C05458=1043.474,385.726,371.742,173.657,43.122,158.451
C05459=1043.465,385.481,371.783,173.649,43.117,158.449
C05460=1043.457,385.234,371.825,173.642,43.112,158.447
C05461=1043.448,384.988,371.867,173.634,43.107,158.445
C05462=1043.439,384.741,371.909,173.627,43.102,158.444
C05463=1043.432,384.495,371.951,173.621,43.097,158.442
C05464=1043.423,384.249,371.992,173.614,43.091,158.440
C05465=1043.414,384.003,372.034,173.606,43.086,158.438
C05466=1043.406,383.757,372.076,173.599,43.082,158.436
C05467=1043.397,383.510,372.118,173.592,43.077,158.435
C05468=1043.389,383.263,372.159,173.584,43.071,158.433
C05469=1043.380,383.018,372.200,173.577,43.066,158.431
C05470=1043.371,382.771,372.242,173.571,43.061,158.429
C05471=1043.363,382.524,372.284,173.564,43.056,158.427
C05472=1043.355,382.278,372.325,173.557,43.052,158.426
C05473=1043.346,382.032,372.367,173.549,43.047,158.424
C05474=1043.338,381.786,372.407,173.542,43.042,158.422
C05475=1043.330,381.539,372.450,173.536,43.037,158.420
C05476=1043.322,381.293,372.491,173.529,43.032,158.419
C05477=1043.313,381.046,372.532,173.521,43.027,158.417
C05478=1043.305,380.801,372.573,173.514,43.022,158.415
C05479=1043.297,380.553,372.615,173.507,43.017,158.413
C05480=1043.289,380.308,372.656,173.501,43.012,158.412
C05481=1043.280,380.061,372.697,173.494,43.007,158.410
C05482=1043.272,379.814,372.738,173.486,43.002,158.408
C05483=1043.264,379.569,372.779,173.480,42.997,158.406
C05484=1043.256,379.321,372.821,173.473,42.992,158.405
C05485=1043.248,379.075,372.861,173.466,42.988,158.403
C05486=1043.239,378.829,372.903,173.460,42.983,158.401
C05487=1043.231,378.582,372.944,173.453,42.978,158.400
C05488=1043.223,378.336,372.984,173.446,42.974,158.398
C05489=1043.214,378.089,373.025,173.438,42.969,158.396
C05490=1043.205,377.843,373.065,173.432,42.964,158.395
C05491=1043.197,377.596,373.106,173.425,42.959,158.393
C05492=1043.189,377.350,373.147,173.418,42.955,158.391
C05493=1043.176,376.988,373.207,173.409,42.948,158.389
C05494=1043.165,376.627,373.267,173.399,42.941,158.386
C05495=1043.153,376.264,373.326,173.389,42.934,158.384
C05496=1043.140,375.903,373.386,173.379,42.928,158.382
C05497=1043.132,375.656,373.426,173.373,42.923,158.380
C05498=1043.124,375.410,373.467,173.366,42.919,158.378
C05499=1043.116,375.163,373.507,173.360,42.914,158.377
C05500=1043.107,374.916,373.548,173.353,42.909,158.375
C05501=1043.099,374.670,373.589,173.346,42.905,158.373
C05502=1043.092,374.423,373.629,173.340,42.900,158.372
C05503=1043.083,374.177,373.669,173.333,42.896,158.370
C05504=1043.075,373.931,373.710,173.327,42.891,158.369
C05505=1043.067,373.684,373.749,173.320,42.887,158.367
C05506=1043.058,373.437,373.790,173.314,42.882,158.365
C05507=1043.051,373.190,373.830,173.307,42.877,158.364
C05508=1043.043,372.944,373.871,173.301,42.873,158.362
C05509=1043.035,372.697,373.912,173.294,42.869,158.361
C05510=1043.026,372.451,373.951,173.288,42.864,158.359
C05511=1043.018,372.205,373.992,173.281,42.860,158.358
C05512=1043.010,371.958,374.032,173.275,42.855,158.356
C05513=1043.003,371.711,374.071,173.268,42.851,158.354
C05514=1042.995,371.465,374.112,173.262,42.846,158.353
C05515=1042.987,371.218,374.152,173.257,42.842,158.351
C05516=1042.978,370.972,374.192,173.250,42.838,158.350
C05517=1042.971,370.725,374.232,173.244,42.833,158.348
C05518=1042.963,370.478,374.272,173.237,42.829,158.347
C05519=1042.954,370.231,374.311,173.231,42.824,158.345
C05520=1042.947,369.984,374.351,173.224,42.821,158.344
C05521=1042.939,369.738,374.392,173.218,42.816,158.342
C05522=1042.930,369.491,374.431,173.212,42.812,158.341
C05523=1042.922,369.245,374.471,173.205,42.808,158.339
C05524=1042.914,368.998,374.510,173.199,42.803,158.338
C05525=1042.906,368.751,374.550,173.193,42.799,158.336
C05526=1042.898,368.504,374.590,173.187,42.795,158.335
C05527=1042.890,368.258,374.629,173.181,42.791,158.333
C05528=1042.882,368.011,374.669,173.174,42.786,158.332
C05529=1042.874,367.764,374.709,173.168,42.782,158.330
C05530=1042.866,367.518,374.748,173.162,42.778,158.329
C05531=1042.858,367.271,374.788,173.156,42.774,158.327
C05532=1042.850,367.024,374.826,173.150,42.769,158.326
C05533=1042.842,366.777,374.866,173.143,42.766,158.325
C05534=1042.834,366.531,374.905,173.137,42.762,158.323
C05535=1042.826,366.284,374.945,173.131,42.757,158.322
C05536=1042.818,366.038,374.984,173.126,42.753,158.320
C05537=1042.811,365.790,375.024,173.119,42.749,158.319
C05538=1042.803,365.544,375.063,173.113,42.745,158.317
C05539=1042.795,365.297,375.103,173.107,42.741,158.316
C05540=1042.787,365.051,375.142,173.101,42.737,158.314
C05541=1042.780,364.803,375.181,173.095,42.732,158.313
C05542=1042.771,364.557,375.220,173.089,42.728,158.312
C05543=1042.764,364.310,375.259,173.083,42.724,158.310
C05544=1042.756,364.063,375.298,173.077,42.721,158.309
C05545=1042.748,363.816,375.338,173.071,42.717,158.307
C05546=1042.741,363.570,375.377,173.065,42.713,158.306
C05547=1042.733,363.323,375.416,173.059,42.708,158.304
C05548=1042.725,363.076,375.455,173.054,42.704,158.303
C05549=1042.714,362.733,375.509,173.045,42.698,158.301
C05550=1042.704,362.392,375.564,173.037,42.693,158.299
C05551=1042.693,362.050,375.617,173.029,42.688,158.297
C05552=1042.682,361.707,375.671,173.020,42.682,158.295
C05553=1042.674,361.461,375.709,173.014,42.678,158.294
C05554=1042.666,361.214,375.749,173.009,42.674,158.293
C05555=1042.658,360.967,375.787,173.003,42.670,158.291
C05556=1042.651,360.720,375.826,172.998,42.667,158.290
C05557=1042.643,360.473,375.865,172.992,42.663,158.289
C05558=1042.635,360.226,375.903,172.985,42.659,158.287
C05559=1042.627,359.979,375.942,172.979,42.655,158.286
C05560=1042.619,359.733,375.981,172.974,42.651,158.285
C05561=1042.612,359.486,376.020,172.968,42.647,158.283
C05562=1042.604,359.239,376.058,172.963,42.643,158.282
C05563=1042.596,358.992,376.097,172.957,42.639,158.281
C05564=1042.588,358.745,376.135,172.951,42.636,158.279
C05565=1042.580,358.498,376.174,172.946,42.632,158.278
C05566=1042.573,358.252,376.212,172.939,42.628,158.277
C05567=1042.565,358.004,376.250,172.934,42.625,158.275
C05568=1042.558,357.757,376.289,172.928,42.621,158.274
C05569=1042.550,357.510,376.327,172.922,42.617,158.273
C05570=1042.542,357.263,376.365,172.917,42.613,158.271
C05571=1042.535,357.017,376.404,172.911,42.610,158.270
C05572=1042.527,356.770,376.442,172.906,42.606,158.269
C05573=1042.519,356.523,376.480,172.900,42.602,158.268
C05574=1042.511,356.275,376.518,172.894,42.598,158.266
C05575=1042.504,356.029,376.557,172.889,42.595,158.265
C05576=1042.496,355.782,376.595,172.883,42.591,158.264
C05577=1042.488,355.534,376.633,172.878,42.587,158.262
C05578=1042.481,355.288,376.671,172.872,42.584,158.261
C05579=1042.473,355.041,376.709,172.867,42.580,158.260
C05580=1042.465,354.793,376.747,172.861,42.576,158.259
C05581=1042.458,354.547,376.785,172.856,42.573,158.257
C05582=1042.451,354.300,376.823,172.850,42.569,158.256
C05583=1042.442,354.053,376.861,172.844,42.565,158.255
C05584=1042.435,353.805,376.899,172.839,42.562,158.254
C05585=1042.428,353.559,376.937,172.834,42.558,158.252
C05586=1042.420,353.312,376.974,172.828,42.555,158.251
C05587=1042.412,353.065,377.013,172.822,42.551,158.250
C05588=1042.404,352.818,377.050,172.817,42.547,158.249
C05589=1042.397,352.571,377.088,172.811,42.544,158.247
C05590=1042.390,352.324,377.126,172.806,42.540,158.246
C05591=1042.382,352.077,377.164,172.801,42.537,158.245
C05592=1042.374,351.829,377.202,172.795,42.533,158.244
C05593=1042.367,351.583,377.240,172.789,42.529,158.242
C05594=1042.360,351.335,377.277,172.784,42.526,158.241
C05595=1042.352,351.088,377.315,172.778,42.522,158.240
C05596=1042.345,350.842,377.353,172.773,42.519,158.239
C05597=1042.337,350.595,377.390,172.769,42.515,158.238
C05598=1042.330,350.348,377.428,172.763,42.512,158.236
C05599=1042.322,350.100,377.465,172.758,42.508,158.235
C05600=1042.315,349.853,377.503,172.752,42.505,158.234
C05601=1042.307,349.606,377.540,172.747,42.501,158.233
C05602=1042.299,349.359,377.577,172.741,42.498,158.232
C05603=1042.292,349.112,377.615,172.736,42.495,158.231
C05604=1042.285,348.865,377.652,172.730,42.492,158.229
C05605=1042.274,348.529,377.703,172.723,42.486,158.228
C05606=1042.264,348.192,377.754,172.717,42.482,158.226
C05607=1042.254,347.857,377.805,172.710,42.477,158.225
C05608=1042.243,347.519,377.856,172.702,42.473,158.223
C05609=1042.236,347.272,377.893,172.697,42.469,158.222
C05610=1042.228,347.025,377.930,172.692,42.466,158.221
C05611=1042.221,346.778,377.968,172.687,42.463,158.220
C05612=1042.214,346.530,378.005,172.681,42.460,158.218
C05613=1042.206,346.284,378.041,172.676,42.456,158.217
C05614=1042.199,346.037,378.079,172.671,42.452,158.216
C05615=1042.191,345.790,378.116,172.666,42.450,158.215
C05616=1042.184,345.543,378.153,172.661,42.446,158.214
C05617=1042.177,345.295,378.190,172.655,42.443,158.213
C05618=1042.169,345.049,378.227,172.650,42.440,158.212
C05619=1042.162,344.802,378.264,172.645,42.436,158.210
C05620=1042.154,344.554,378.301,172.640,42.433,158.209
C05621=1042.147,344.307,378.338,172.635,42.430,158.208
C05622=1042.139,344.059,378.374,172.629,42.427,158.207
C05623=1042.132,343.812,378.412,172.625,42.423,158.206
C05624=1042.125,343.565,378.449,172.620,42.420,158.205
C05625=1042.118,343.318,378.485,172.614,42.417,158.204
C05626=1042.110,343.071,378.523,172.609,42.414,158.203
C05627=1042.103,342.824,378.559,172.605,42.410,158.201
C05628=1042.096,342.576,378.596,172.599,42.407,158.200
C05629=1042.088,342.329,378.633,172.594,42.404,158.199
C05630=1042.082,342.082,378.669,172.590,42.401,158.198
C05631=1042.074,341.835,378.706,172.585,42.398,158.197
C05632=1042.067,341.588,378.743,172.579,42.394,158.196
C05633=1042.059,341.340,378.779,172.574,42.391,158.195
C05634=1042.051,341.093,378.816,172.570,42.388,158.194
C05635=1042.044,340.846,378.853,172.564,42.385,158.193
C05636=1042.037,340.599,378.889,172.559,42.382,158.192
C05637=1042.029,340.351,378.925,172.555,42.379,158.191
C05638=1042.021,340.105,378.962,172.549,42.376,158.190
C05639=1042.014,339.857,378.999,172.544,42.372,158.188
C05640=1042.007,339.610,379.035,172.540,42.369,158.187
C05641=1042.000,339.363,379.071,172.535,42.366,158.186
C05642=1041.993,339.115,379.108,172.529,42.363,158.185
C05643=1041.986,338.868,379.143,172.525,42.360,158.184
C05644=1041.978,338.621,379.180,172.520,42.357,158.183
C05645=1041.970,338.374,379.217,172.514,42.354,158.182
C05646=1041.964,338.127,379.253,172.510,42.351,158.181
C05647=1041.956,337.879,379.289,172.505,42.348,158.180
C05648=1041.948,337.632,379.325,172.500,42.345,158.179
C05649=1041.942,337.385,379.362,172.495,42.342,158.178
C05650=1041.934,337.137,379.398,172.490,42.339,158.177
C05651=1041.927,336.890,379.434,172.486,42.336,158.176
C05652=1041.919,336.643,379.470,172.481,42.333,158.175
C05653=1041.913,336.396,379.507,172.476,42.330,158.174
C05654=1041.906,336.148,379.542,172.471,42.327,158.173
C05655=1041.898,335.901,379.578,172.466,42.324,158.172
C05656=1041.890,335.653,379.615,172.462,42.321,158.171
C05657=1041.884,335.406,379.651,172.457,42.318,158.170
C05658=1041.876,335.159,379.687,172.452,42.315,158.169
C05659=1041.869,334.912,379.723,172.447,42.312,158.168
C05660=1041.862,334.664,379.759,172.442,42.309,158.167
C05661=1041.852,334.324,379.808,172.435,42.305,158.165
C05662=1041.842,333.984,379.857,172.430,42.301,158.164
C05663=1041.832,333.644,379.906,172.423,42.297,158.163
C05664=1041.822,333.304,379.956,172.416,42.293,158.161
C05665=1041.815,333.057,379.991,172.411,42.290,158.160
C05666=1041.808,332.809,380.027,172.407,42.287,158.159
C05667=1041.800,332.563,380.063,172.402,42.284,158.158
C05668=1041.793,332.315,380.098,172.398,42.281,158.157
C05669=1041.786,332.068,380.134,172.393,42.278,158.156
C05670=1041.778,331.820,380.170,172.388,42.275,158.155
C05671=1041.772,331.573,380.205,172.383,42.273,158.154
C05672=1041.764,331.325,380.241,172.379,42.270,158.153
C05673=1041.757,331.078,380.277,172.374,42.267,158.152
C05674=1041.750,330.831,380.312,172.370,42.264,158.152
C05675=1041.743,330.583,380.348,172.365,42.261,158.151
C05676=1041.736,330.336,380.383,172.360,42.258,158.150
C05677=1041.728,330.089,380.420,172.355,42.256,158.149
C05678=1041.722,329.841,380.455,172.351,42.253,158.148
C05679=1041.715,329.594,380.490,172.346,42.250,158.147
C05680=1041.707,329.346,380.526,172.342,42.247,158.146
C05681=1041.700,329.099,380.561,172.338,42.244,158.145
C05682=1041.693,328.852,380.596,172.333,42.241,158.144
C05683=1041.685,328.604,380.631,172.328,42.239,158.143
C05684=1041.678,328.357,380.667,172.323,42.236,158.142
C05685=1041.670,328.109,380.702,172.319,42.233,158.141
C05686=1041.663,327.862,380.737,172.314,42.231,158.140
C05687=1041.656,327.615,380.772,172.310,42.228,158.139
C05688=1041.649,327.367,380.807,172.305,42.225,158.138
C05689=1041.642,327.120,380.842,172.301,42.223,158.137
C05690=1041.634,326.873,380.877,172.296,42.220,158.136
C05691=1041.627,326.624,380.912,172.292,42.217,158.136
C05692=1041.619,326.377,380.947,172.287,42.215,158.135
C05693=1041.613,326.130,380.982,172.283,42.212,158.134
C05694=1041.605,325.882,381.017,172.279,42.209,158.133
C05695=1041.598,325.635,381.052,172.274,42.207,158.132
C05696=1041.591,325.388,381.087,172.269,42.204,158.131
C05697=1041.584,325.140,381.122,172.264,42.201,158.130
C05698=1041.576,324.892,381.157,172.260,42.199,158.129
C05699=1041.569,324.645,381.192,172.256,42.196,158.128
C05700=1041.562,324.398,381.227,172.251,42.193,158.127
C05701=1041.554,324.151,381.261,172.247,42.191,158.127
C05702=1041.548,323.903,381.296,172.242,42.188,158.126
C05703=1041.541,323.655,381.331,172.238,42.185,158.125
C05704=1041.533,323.408,381.366,172.234,42.183,158.124
C05705=1041.526,323.160,381.401,172.229,42.180,158.123
C05706=1041.519,322.913,381.436,172.225,42.178,158.122
C05707=1041.512,322.665,381.470,172.221,42.175,158.121
C05708=1041.505,322.418,381.504,172.216,42.172,158.120
C05709=1041.497,322.170,381.540,172.212,42.170,158.119
C05710=1041.490,321.923,381.575,172.208,42.167,158.119
C05711=1041.483,321.675,381.609,172.203,42.165,158.118
C05712=1041.476,321.428,381.643,172.199,42.162,158.117
C05713=1041.469,321.181,381.679,172.195,42.160,158.116
C05714=1041.462,320.933,381.712,172.189,42.157,158.115
C05715=1041.455,320.686,381.748,172.185,42.154,158.114
C05716=1041.448,320.438,381.781,172.181,42.152,158.113
C05717=1041.438,320.094,381.831,172.175,42.148,158.112
C05718=1041.428,319.749,381.879,172.170,42.145,158.111
C05719=1041.418,319.404,381.927,172.163,42.141,158.110
C05720=1041.409,319.059,381.975,172.157,42.138,158.108
C05721=1041.402,318.811,382.009,172.153,42.135,158.108
C05722=1041.395,318.564,382.044,172.149,42.133,158.107
C05723=1041.388,318.316,382.078,172.145,42.130,158.106
C05724=1041.381,318.069,382.113,172.140,42.128,158.105
C05725=1041.375,317.822,382.146,172.136,42.125,158.104
C05726=1041.368,317.574,382.182,172.132,42.123,158.103
C05727=1041.361,317.327,382.215,172.128,42.120,158.103
C05728=1041.353,317.079,382.249,172.123,42.118,158.102
C05729=1041.347,316.832,382.284,172.119,42.115,158.101
C05730=1041.339,316.584,382.318,172.115,42.113,158.100
C05731=1041.333,316.337,382.353,172.111,42.110,158.099
C05732=1041.326,316.089,382.387,172.107,42.108,158.098
C05733=1041.319,315.841,382.422,172.102,42.105,158.097
C05734=1041.312,315.593,382.455,172.098,42.103,158.097
C05735=1041.306,315.347,382.490,172.094,42.100,158.096
C05736=1041.298,315.099,382.524,172.090,42.098,158.095
C05737=1041.292,314.851,382.558,172.086,42.095,158.094
C05738=1041.285,314.604,382.593,172.081,42.093,158.093
C05739=1041.278,314.356,382.627,172.077,42.090,158.092
C05740=1041.271,314.109,382.661,172.073,42.088,158.092
C05741=1041.265,313.861,382.695,172.069,42.085,158.091
C05742=1041.258,313.613,382.729,172.065,42.083,158.090
C05743=1041.251,313.366,382.763,172.061,42.080,158.089
C05744=1041.244,313.119,382.798,172.056,42.078,158.088
C05745=1041.237,312.871,382.831,172.052,42.075,158.087
C05746=1041.231,312.623,382.866,172.048,42.073,158.087
C05747=1041.224,312.376,382.900,172.044,42.070,158.086
C05748=1041.217,312.129,382.933,172.040,42.068,158.085
C05749=1041.210,311.881,382.967,172.036,42.066,158.084
C05750=1041.203,311.633,383.001,172.031,42.063,158.083
C05751=1041.195,311.386,383.035,172.027,42.062,158.083
C05752=1041.188,311.138,383.068,172.023,42.059,158.082
C05753=1041.181,310.890,383.102,172.020,42.057,158.081
C05754=1041.175,310.643,383.135,172.016,42.054,158.080
C05755=1041.167,310.395,383.169,172.012,42.052,158.080
C05756=1041.160,310.147,383.203,172.007,42.050,158.079
C05757=1041.150,309.818,383.247,172.002,42.047,158.078
C05758=1041.141,309.488,383.292,171.997,42.044,158.077
C05759=1041.131,309.159,383.336,171.991,42.041,158.076
C05760=1041.123,308.829,383.380,171.986,42.038,158.075
C05761=1041.116,308.581,383.414,171.982,42.035,158.074
C05762=1041.108,308.334,383.448,171.977,42.034,158.073
C05763=1041.102,308.086,383.480,171.973,42.031,158.072
C05764=1041.095,307.838,383.514,171.970,42.029,158.072
C05765=1041.087,307.591,383.547,171.966,42.027,158.071
C05766=1041.080,307.343,383.581,171.962,42.025,158.070
C05767=1041.073,307.096,383.614,171.958,42.022,158.069
C05768=1041.066,306.848,383.648,171.954,42.020,158.069
C05769=1041.060,306.600,383.681,171.950,42.018,158.068
C05770=1041.053,306.353,383.714,171.946,42.015,158.067
C05771=1041.045,306.105,383.747,171.941,42.014,158.066
C05772=1041.038,305.858,383.780,171.937,42.011,158.066
C05773=1041.031,305.599,383.815,171.934,42.009,158.065
C05774=1041.024,305.341,383.850,171.930,42.007,158.064
C05775=1041.017,305.084,383.884,171.926,42.004,158.063
C05776=1041.010,304.825,383.919,171.922,42.002,158.063
C05777=1041.003,304.578,383.952,171.918,42.000,158.062
C05778=1040.996,304.330,383.985,171.914,41.997,158.061
C05779=1040.990,304.082,384.018,171.909,41.996,158.060
C05780=1040.982,303.835,384.051,171.905,41.993,158.059
C05781=1040.976,303.587,384.084,171.902,41.991,158.059
C05782=1040.968,303.340,384.118,171.898,41.989,158.058
C05783=1040.961,303.091,384.151,171.894,41.987,158.057
C05784=1040.955,302.844,384.184,171.890,41.985,158.057
C05785=1040.948,302.597,384.217,171.886,41.983,158.056
C05786=1040.941,302.349,384.250,171.882,41.980,158.055
C05787=1040.935,302.101,384.282,171.878,41.978,158.054
C05788=1040.927,301.854,384.316,171.875,41.976,158.054
C05789=1040.921,301.606,384.349,171.871,41.974,158.053
C05790=1040.914,301.358,384.382,171.867,41.972,158.052
C05791=1040.907,301.110,384.414,171.863,41.970,158.051
C05792=1040.900,300.863,384.448,171.859,41.967,158.051
C05793=1040.894,300.615,384.481,171.855,41.965,158.050
C05794=1040.887,300.367,384.514,171.852,41.963,158.049
C05795=1040.880,300.120,384.546,171.849,41.960,158.048
C05796=1040.873,299.872,384.579,171.845,41.958,158.048
C05797=1040.866,299.624,384.613,171.841,41.956,158.047
C05798=1040.860,299.377,384.645,171.837,41.954,158.046
C05799=1040.854,299.129,384.678,171.833,41.952,158.046
C05800=1040.846,298.881,384.711,171.829,41.950,158.045
C05801=1040.840,298.634,384.743,171.826,41.948,158.044
C05802=1040.833,298.386,384.776,171.822,41.946,158.044
C05803=1040.827,298.138,384.809,171.818,41.943,158.043
C05804=1040.820,297.890,384.841,171.814,41.941,158.042
C05805=1040.813,297.643,384.874,171.810,41.939,158.041
C05806=1040.806,297.394,384.907,171.807,41.937,158.041
C05807=1040.800,297.147,384.940,171.803,41.935,158.040
C05808=1040.794,296.899,384.973,171.799,41.933,158.039
C05809=1040.786,296.651,385.005,171.796,41.931,158.039
C05810=1040.780,296.404,385.038,171.792,41.929,158.038
C05811=1040.774,296.156,385.071,171.788,41.927,158.037
C05812=1040.767,295.909,385.103,171.784,41.924,158.036
C05813=1040.760,295.661,385.136,171.781,41.922,158.036
C05814=1040.753,295.413,385.169,171.777,41.920,158.035
C05815=1040.747,295.165,385.201,171.773,41.918,158.034
C05816=1040.739,294.917,385.234,171.769,41.916,158.034
C05817=1040.733,294.669,385.265,171.766,41.914,158.033
C05818=1040.726,294.422,385.298,171.763,41.912,158.032
C05819=1040.719,294.175,385.330,171.759,41.910,158.032
C05820=1040.712,293.926,385.363,171.755,41.908,158.031
C05821=1040.706,293.678,385.395,171.751,41.906,158.030
C05822=1040.699,293.431,385.428,171.748,41.904,158.030
C05823=1040.692,293.183,385.460,171.744,41.902,158.029
C05824=1040.685,292.935,385.492,171.740,41.900,158.028
C05825=1040.679,292.687,385.524,171.736,41.898,158.028
C05826=1040.672,292.440,385.556,171.734,41.896,158.027
C05827=1040.664,292.191,385.588,171.730,41.894,158.026
C05828=1040.658,291.944,385.621,171.726,41.892,158.026
C05829=1040.649,291.621,385.663,171.721,41.889,158.025
C05830=1040.640,291.296,385.705,171.716,41.887,158.024
C05831=1040.631,290.973,385.746,171.712,41.884,158.023
C05832=1040.623,290.650,385.788,171.707,41.882,158.022
C05833=1040.616,290.402,385.820,171.703,41.880,158.021
C05834=1040.609,290.155,385.852,171.700,41.878,158.021
C05835=1040.603,289.906,385.884,171.696,41.876,158.020
C05836=1040.596,289.658,385.916,171.693,41.874,158.019
C05837=1040.589,289.411,385.948,171.689,41.872,158.019
C05838=1040.582,289.163,385.980,171.685,41.870,158.018
C05839=1040.575,288.915,386.013,171.682,41.868,158.018
C05840=1040.569,288.667,386.044,171.678,41.866,158.017
C05841=1040.562,288.419,386.075,171.675,41.864,158.016
C05842=1040.555,288.172,386.108,171.672,41.862,158.016
C05843=1040.549,287.924,386.140,171.668,41.860,158.015
C05844=1040.542,287.676,386.172,171.664,41.858,158.014
C05845=1040.535,287.428,386.203,171.660,41.857,158.014
C05846=1040.528,287.180,386.235,171.658,41.855,158.013
C05847=1040.521,286.932,386.266,171.654,41.853,158.012
C05848=1040.514,286.685,386.299,171.650,41.851,158.012
C05849=1040.507,286.437,386.330,171.646,41.849,158.011
C05850=1040.501,286.189,386.362,171.643,41.847,158.010
C05851=1040.495,285.941,386.393,171.640,41.845,158.010
C05852=1040.488,285.693,386.425,171.636,41.843,158.009
C05853=1040.481,285.446,386.457,171.633,41.842,158.009
C05854=1040.474,285.198,386.488,171.629,41.840,158.008
C05855=1040.467,284.949,386.520,171.626,41.838,158.007
C05856=1040.460,284.701,386.552,171.622,41.836,158.007
C05857=1040.453,284.453,386.583,171.619,41.834,158.006
C05858=1040.447,284.205,386.615,171.615,41.832,158.005
C05859=1040.440,283.957,386.646,171.612,41.831,158.005
C05860=1040.433,283.709,386.677,171.609,41.829,158.004
C05861=1040.426,283.462,386.709,171.605,41.827,158.004
C05862=1040.420,283.214,386.740,171.601,41.825,158.003
C05863=1040.413,282.966,386.772,171.598,41.823,158.002
C05864=1040.406,282.718,386.803,171.595,41.821,158.002
C05865=1040.400,282.470,386.835,171.591,41.820,158.001
C05866=1040.393,282.222,386.866,171.587,41.818,158.001
C05867=1040.386,281.974,386.897,171.585,41.816,158.000
C05868=1040.379,281.726,386.929,171.581,41.814,157.999
C05869=1040.373,281.478,386.960,171.577,41.812,157.999
C05870=1040.366,281.230,386.992,171.574,41.810,157.998
C05871=1040.359,280.983,387.023,171.571,41.809,157.998
C05872=1040.352,280.735,387.055,171.567,41.807,157.997
C05873=1040.346,280.487,387.086,171.564,41.804,157.996
C05874=1040.339,280.239,387.117,171.561,41.803,157.996
C05875=1040.333,279.991,387.148,171.557,41.801,157.995
C05876=1040.326,279.743,387.179,171.553,41.800,157.994
C05877=1040.320,279.495,387.211,171.551,41.798,157.994
C05878=1040.313,279.247,387.242,171.547,41.796,157.993
C05879=1040.306,279.000,387.273,171.543,41.794,157.993
C05880=1040.299,278.752,387.304,171.540,41.792,157.992
C05881=1040.292,278.503,387.335,171.537,41.791,157.991
C05882=1040.286,278.255,387.366,171.533,41.789,157.991
C05883=1040.279,278.007,387.398,171.531,41.787,157.990
C05884=1040.273,277.759,387.429,171.527,41.785,157.990
C05885=1040.264,277.448,387.467,171.523,41.783,157.989
C05886=1040.255,277.136,387.506,171.518,41.780,157.988
C05887=1040.247,276.825,387.545,171.514,41.778,157.987
C05888=1040.239,276.513,387.584,171.510,41.776,157.987
C05889=1040.232,276.265,387.616,171.507,41.774,157.986
C05890=1040.225,276.017,387.646,171.504,41.772,157.985
C05891=1040.218,275.769,387.677,171.500,41.771,157.985
C05892=1040.212,275.521,387.708,171.497,41.769,157.984
C05893=1040.205,275.273,387.739,171.494,41.767,157.984
C05894=1040.198,275.025,387.769,171.490,41.766,157.983
C05895=1040.192,274.777,387.801,171.487,41.764,157.983
C05896=1040.185,274.529,387.831,171.484,41.762,157.982
C05897=1040.178,274.281,387.862,171.480,41.760,157.981
C05898=1040.171,274.033,387.893,171.478,41.759,157.981
C05899=1040.165,273.785,387.924,171.474,41.757,157.980
C05900=1040.158,273.537,387.954,171.470,41.755,157.980
C05901=1040.151,273.289,387.986,171.468,41.754,157.979
C05902=1040.145,273.041,388.016,171.464,41.752,157.979
C05903=1040.138,272.793,388.046,171.462,41.750,157.978
C05904=1040.131,272.545,388.078,171.458,41.748,157.977
C05905=1040.125,272.297,388.108,171.454,41.747,157.977
C05906=1040.118,272.049,388.139,171.451,41.745,157.976
C05907=1040.111,271.801,388.170,171.448,41.743,157.976
C05908=1040.104,271.553,388.200,171.445,41.742,157.975
C05909=1040.098,271.305,388.231,171.442,41.740,157.975
C05910=1040.092,271.057,388.262,171.438,41.738,157.974
C05911=1040.085,270.809,388.292,171.435,41.737,157.973
C05912=1040.078,270.560,388.322,171.432,41.735,157.973
C05913=1040.071,270.313,388.353,171.429,41.733,157.972
C05914=1040.065,270.065,388.384,171.425,41.732,157.972
C05915=1040.058,269.816,388.414,171.423,41.729,157.971
C05916=1040.051,269.568,388.444,171.419,41.728,157.971
C05917=1040.045,269.320,388.474,171.417,41.726,157.970
C05918=1040.037,269.073,388.505,171.413,41.724,157.969
C05919=1040.031,268.824,388.536,171.409,41.723,157.969
C05920=1040.024,268.577,388.566,171.407,41.721,157.968
C05921=1040.018,268.328,388.596,171.403,41.719,157.968
C05922=1040.011,268.080,388.626,171.400,41.718,157.967
C05923=1040.005,267.832,388.657,171.397,41.716,157.967
C05924=1039.998,267.584,388.687,171.394,41.715,157.966
C05925=1039.991,267.335,388.718,171.390,41.713,157.966
C05926=1039.985,267.089,388.748,171.388,41.711,157.965
C05927=1039.977,266.840,388.778,171.384,41.710,157.965
C05928=1039.971,266.592,388.809,171.382,41.708,157.964
C05929=1039.964,266.344,388.839,171.378,41.706,157.963
C05930=1039.957,266.096,388.869,171.375,41.705,157.963
C05931=1039.951,265.848,388.899,171.372,41.703,157.962
C05932=1039.944,265.600,388.929,171.369,41.702,157.962
C05933=1039.937,265.351,388.959,171.365,41.700,157.961
C05934=1039.931,265.103,388.989,171.363,41.698,157.961
C05935=1039.924,264.855,389.019,171.359,41.697,157.960
C05936=1039.917,264.607,389.049,171.357,41.695,157.960
C05937=1039.911,264.358,389.080,171.353,41.693,157.959
C05938=1039.904,264.111,389.110,171.350,41.692,157.959
C05939=1039.897,263.863,389.140,171.347,41.690,157.958
C05940=1039.891,263.615,389.170,171.344,41.689,157.958
C05941=1039.883,263.308,389.207,171.340,41.687,157.957
C05942=1039.874,263.000,389.245,171.337,41.685,157.956
C05943=1039.866,262.693,389.282,171.333,41.683,157.956
C05944=1039.858,262.386,389.319,171.329,41.680,157.955
C05945=1039.852,262.138,389.348,171.326,41.679,157.954
C05946=1039.845,261.890,389.378,171.323,41.677,157.954
C05947=1039.838,261.642,389.409,171.319,41.676,157.953
C05948=1039.831,261.394,389.438,171.317,41.674,157.953
C05949=1039.824,261.146,389.468,171.313,41.672,157.952
C05950=1039.818,260.898,389.497,171.311,41.671,157.952
C05951=1039.811,260.649,389.527,171.307,41.669,157.951
C05952=1039.804,260.401,389.557,171.304,41.668,157.951
C05953=1039.797,260.153,389.586,171.301,41.666,157.950
C05954=1039.790,259.905,389.616,171.298,41.665,157.950
C05955=1039.784,259.657,389.646,171.295,41.663,157.949
C05956=1039.776,259.409,389.675,171.292,41.662,157.949
C05957=1039.769,259.161,389.704,171.289,41.660,157.948
C05958=1039.763,258.912,389.734,171.286,41.659,157.948
C05959=1039.755,258.664,389.764,171.283,41.657,157.947
C05960=1039.749,258.416,389.793,171.280,41.656,157.947
C05961=1039.742,258.168,389.823,171.277,41.654,157.946
C05962=1039.736,257.920,389.852,171.274,41.653,157.946
C05963=1039.729,257.671,389.882,171.271,41.651,157.945
C05964=1039.722,257.423,389.911,171.268,41.650,157.945
C05965=1039.715,257.175,389.941,171.265,41.648,157.944
C05966=1039.709,256.927,389.971,171.262,41.647,157.944
C05967=1039.702,256.679,390.001,171.259,41.645,157.943
C05968=1039.695,256.431,390.029,171.256,41.644,157.943
C05969=1039.688,256.182,390.059,171.253,41.642,157.942
C05970=1039.681,255.934,390.088,171.250,41.641,157.942
C05971=1039.675,255.686,390.118,171.248,41.639,157.941
C05972=1039.668,255.438,390.147,171.244,41.638,157.941
C05973=1039.662,255.190,390.176,171.242,41.636,157.940
C05974=1039.655,254.941,390.206,171.238,41.635,157.940
C05975=1039.648,254.694,390.236,171.235,41.633,157.939
C05976=1039.641,254.445,390.265,171.233,41.632,157.939
C05977=1039.635,254.197,390.294,171.229,41.630,157.938
C05978=1039.627,253.949,390.324,171.227,41.629,157.938
C05979=1039.621,253.701,390.353,171.224,41.627,157.937
C05980=1039.615,253.453,390.382,171.221,41.626,157.937
C05981=1039.608,253.204,390.412,171.218,41.624,157.936
C05982=1039.601,252.956,390.441,171.215,41.623,157.936
C05983=1039.595,252.707,390.470,171.212,41.621,157.935
C05984=1039.588,252.459,390.499,171.209,41.619,157.935
C05985=1039.582,252.212,390.529,171.207,41.618,157.934
C05986=1039.574,251.963,390.558,171.203,41.616,157.934
C05987=1039.568,251.715,390.587,171.201,41.615,157.933
C05988=1039.562,251.467,390.616,171.198,41.613,157.933
C05989=1039.555,251.218,390.645,171.194,41.612,157.932
C05990=1039.548,250.971,390.675,171.192,41.610,157.932
C05991=1039.542,250.722,390.704,171.189,41.609,157.931
C05992=1039.535,250.474,390.734,171.186,41.607,157.931
C05993=1039.529,250.225,390.763,171.183,41.606,157.930
C05994=1039.522,249.978,390.791,171.181,41.604,157.930
C05995=1039.515,249.729,390.820,171.177,41.603,157.929
C05996=1039.509,249.481,390.849,171.175,41.601,157.929
C05997=1039.501,249.172,390.886,171.171,41.599,157.928
C05998=1039.493,248.864,390.922,171.167,41.598,157.927
C05999=1039.485,248.556,390.959,171.164,41.595,157.927
C06000=1039.476,248.247,390.995,171.161,41.593,157.926
C06001=1039.470,247.999,391.024,171.158,41.592,157.926
C06002=1039.464,247.751,391.053,171.155,41.590,157.925
C06003=1039.456,247.502,391.082,171.152,41.589,157.925
C06004=1039.450,247.254,391.111,171.149,41.587,157.924
C06005=1039.444,247.006,391.140,171.147,41.586,157.924
C06006=1039.437,246.758,391.169,171.143,41.584,157.923
C06007=1039.431,246.509,391.198,171.141,41.583,157.923
C06008=1039.424,246.261,391.227,171.138,41.581,157.922
C06009=1039.418,246.013,391.257,171.136,41.579,157.922
C06010=1039.411,245.765,391.285,171.132,41.578,157.921
C06011=1039.405,245.517,391.314,171.130,41.576,157.921
C06012=1039.398,245.268,391.343,171.127,41.575,157.920
C06013=1039.392,245.019,391.372,171.124,41.573,157.920
C06014=1039.385,244.771,391.400,171.121,41.572,157.919
C06015=1039.379,244.523,391.429,171.118,41.570,157.919
C06016=1039.373,244.275,391.458,171.116,41.569,157.918
C06017=1039.365,244.027,391.487,171.113,41.568,157.918
C06018=1039.359,243.778,391.516,171.110,41.566,157.917
C06019=1039.352,243.530,391.544,171.107,41.565,157.917
C06020=1039.346,243.282,391.573,171.105,41.563,157.916
C06021=1039.339,243.034,391.601,171.102,41.562,157.916
C06022=1039.332,242.785,391.631,171.100,41.560,157.915
C06023=1039.326,242.536,391.659,171.096,41.558,157.915
C06024=1039.319,242.289,391.688,171.093,41.557,157.914
C06025=1039.313,242.040,391.717,171.091,41.556,157.914
C06026=1039.306,241.793,391.745,171.088,41.554,157.914
C06027=1039.300,241.544,391.773,171.086,41.553,157.913
C06028=1039.293,241.295,391.803,171.082,41.551,157.913
C06029=1039.286,241.047,391.831,171.080,41.550,157.912
C06030=1039.280,240.799,391.859,171.077,41.548,157.912
C06031=1039.273,240.551,391.888,171.075,41.547,157.911
C06032=1039.266,240.302,391.916,171.072,41.546,157.911
C06033=1039.260,240.054,391.945,171.069,41.544,157.910
C06034=1039.253,239.806,391.973,171.066,41.543,157.910
C06035=1039.246,239.557,392.001,171.064,41.541,157.909
C06036=1039.240,239.309,392.030,171.061,41.539,157.909
C06037=1039.233,239.061,392.058,171.059,41.538,157.908
C06038=1039.226,238.813,392.086,171.055,41.537,157.908
C06039=1039.220,238.564,392.115,171.053,41.535,157.907
C06040=1039.213,238.316,392.143,171.050,41.534,157.907
C06041=1039.206,238.068,392.171,171.048,41.533,157.907
C06042=1039.199,237.819,392.200,171.045,41.531,157.906
C06043=1039.193,237.570,392.228,171.042,41.530,157.906
C06044=1039.186,237.323,392.257,171.039,41.528,157.905
C06045=1039.179,237.074,392.284,171.037,41.527,157.905
C06046=1039.173,236.825,392.313,171.034,41.526,157.904
C06047=1039.166,236.578,392.341,171.031,41.524,157.904
C06048=1039.160,236.329,392.369,171.029,41.522,157.903
C06049=1039.153,236.081,392.397,171.026,41.521,157.903
C06050=1039.147,235.833,392.426,171.023,41.520,157.902
C06051=1039.140,235.584,392.453,171.020,41.518,157.902
C06052=1039.133,235.336,392.482,171.018,41.517,157.901
C06053=1039.124,235.022,392.517,171.014,41.515,157.901
C06054=1039.117,234.707,392.553,171.012,41.513,157.900
C06055=1039.108,234.393,392.589,171.008,41.512,157.900
C06056=1039.099,234.078,392.624,171.004,41.510,157.899
C06057=1039.092,233.830,392.652,171.002,41.508,157.899
C06058=1039.086,233.582,392.681,170.999,41.507,157.898
C06059=1039.079,233.333,392.709,170.997,41.506,157.898
C06060=1039.073,233.085,392.737,170.994,41.504,157.897
C06061=1039.066,232.836,392.764,170.992,41.502,157.897
C06062=1039.060,232.588,392.793,170.989,41.501,157.897
C06063=1039.053,232.340,392.821,170.987,41.500,157.896
C06064=1039.046,232.091,392.849,170.984,41.498,157.896
C06065=1039.040,231.843,392.876,170.981,41.497,157.895
C06066=1039.033,231.595,392.905,170.978,41.495,157.895
C06067=1039.026,231.347,392.933,170.976,41.494,157.894
C06068=1039.020,231.098,392.961,170.973,41.493,157.894
C06069=1039.013,230.849,392.989,170.971,41.491,157.893
C06070=1039.007,230.601,393.016,170.968,41.490,157.893
C06071=1039.000,230.353,393.044,170.966,41.488,157.892
C06072=1038.993,230.104,393.072,170.963,41.487,157.892
C06073=1038.987,229.856,393.100,170.961,41.485,157.891
C06074=1038.980,229.608,393.128,170.958,41.484,157.891
C06075=1038.974,229.360,393.155,170.956,41.483,157.891
C06076=1038.967,229.112,393.183,170.953,41.481,157.890
C06077=1038.960,228.863,393.211,170.950,41.480,157.890
C06078=1038.954,228.615,393.239,170.947,41.479,157.889
C06079=1038.948,228.366,393.267,170.945,41.477,157.889
C06080=1038.940,228.118,393.294,170.942,41.475,157.888
C06081=1038.934,227.870,393.322,170.940,41.474,157.888
C06082=1038.927,227.621,393.350,170.937,41.473,157.887
C06083=1038.920,227.373,393.377,170.935,41.472,157.887
C06084=1038.914,227.124,393.405,170.932,41.470,157.887
C06085=1038.907,226.876,393.433,170.930,41.469,157.886
C06086=1038.900,226.627,393.460,170.927,41.468,157.886
C06087=1038.894,226.378,393.487,170.925,41.466,157.885
C06088=1038.886,226.130,393.515,170.922,41.465,157.885
C06089=1038.880,225.882,393.542,170.920,41.464,157.885
C06090=1038.873,225.633,393.570,170.917,41.462,157.884
C06091=1038.867,225.386,393.597,170.915,41.460,157.884
C06092=1038.860,225.137,393.625,170.912,41.459,157.883
C06093=1038.854,224.889,393.653,170.910,41.458,157.883
C06094=1038.847,224.640,393.681,170.907,41.456,157.882
C06095=1038.840,224.391,393.707,170.905,41.455,157.882
C06096=1038.833,224.143,393.735,170.902,41.454,157.881
C06097=1038.826,223.895,393.763,170.900,41.453,157.881
C06098=1038.820,223.646,393.790,170.897,41.451,157.881
C06099=1038.814,223.398,393.818,170.895,41.449,157.880
C06100=1038.807,223.149,393.845,170.892,41.448,157.880
C06101=1038.800,222.901,393.872,170.890,41.447,157.879
C06102=1038.793,222.653,393.900,170.887,41.445,157.879
C06103=1038.787,222.404,393.927,170.885,41.444,157.878
C06104=1038.780,222.155,393.954,170.882,41.443,157.878
C06105=1038.774,221.907,393.982,170.880,41.441,157.878
C06106=1038.767,221.659,394.009,170.878,41.440,157.877
C06107=1038.760,221.411,394.036,170.875,41.438,157.877
C06108=1038.754,221.162,394.063,170.872,41.437,157.876
C06109=1038.746,220.840,394.099,170.869,41.435,157.876
C06110=1038.737,220.518,394.134,170.866,41.433,157.875
C06111=1038.728,220.197,394.169,170.863,41.432,157.875
C06112=1038.720,219.875,394.205,170.860,41.429,157.874
C06113=1038.713,219.627,394.232,170.857,41.428,157.874
C06114=1038.706,219.378,394.259,170.855,41.427,157.873
C06115=1038.699,219.129,394.286,170.853,41.426,157.873
C06116=1038.692,218.881,394.314,170.850,41.424,157.872
C06117=1038.686,218.632,394.341,170.848,41.423,157.872
C06118=1038.679,218.385,394.368,170.845,41.422,157.871
C06119=1038.673,218.135,394.395,170.843,41.420,157.871
C06120=1038.665,217.887,394.422,170.840,41.419,157.871
C06121=1038.659,217.638,394.449,170.838,41.418,157.870
C06122=1038.652,217.391,394.476,170.835,41.417,157.870
C06123=1038.646,217.142,394.503,170.833,41.415,157.869
C06124=1038.639,216.893,394.531,170.830,41.414,157.869
C06125=1038.632,216.645,394.557,170.828,41.412,157.869
C06126=1038.625,216.396,394.585,170.825,41.411,157.868
C06127=1038.619,216.148,394.611,170.823,41.410,157.868
C06128=1038.612,215.899,394.638,170.820,41.408,157.867
C06129=1038.605,215.651,394.665,170.818,41.407,157.867
C06130=1038.599,215.403,394.692,170.815,41.406,157.866
C06131=1038.592,215.154,394.719,170.814,41.404,157.866
C06132=1038.585,214.905,394.746,170.812,41.403,157.866
C06133=1038.578,214.657,394.773,170.809,41.401,157.865
C06134=1038.572,214.409,394.800,170.807,41.400,157.865
C06135=1038.566,214.160,394.827,170.804,41.399,157.864
C06136=1038.558,213.912,394.854,170.802,41.397,157.864
C06137=1038.553,213.663,394.880,170.799,41.396,157.863
C06138=1038.546,213.415,394.907,170.797,41.394,157.863
C06139=1038.539,213.166,394.935,170.794,41.393,157.863
C06140=1038.532,212.918,394.961,170.793,41.392,157.862
C06141=1038.526,212.669,394.988,170.790,41.390,157.862
C06142=1038.519,212.421,395.015,170.788,41.389,157.861
C06143=1038.513,212.173,395.041,170.785,41.388,157.861
C06144=1038.506,211.924,395.068,170.783,41.386,157.860
C06145=1038.499,211.675,395.096,170.780,41.385,157.860
C06146=1038.492,211.427,395.122,170.778,41.383,157.860
C06147=1038.486,211.178,395.149,170.775,41.382,157.859
C06148=1038.479,210.929,395.175,170.774,41.381,157.859
C06149=1038.473,210.682,395.202,170.772,41.380,157.858
C06150=1038.466,210.433,395.229,170.769,41.378,157.858
C06151=1038.459,210.184,395.255,170.766,41.376,157.858
C06152=1038.453,209.936,395.282,170.764,41.375,157.857
C06153=1038.446,209.687,395.308,170.762,41.374,157.857
C06154=1038.439,209.439,395.334,170.759,41.373,157.856
C06155=1038.433,209.191,395.362,170.758,41.371,157.856
C06156=1038.426,208.942,395.388,170.755,41.370,157.856
C06157=1038.419,208.694,395.415,170.753,41.368,157.855
C06158=1038.413,208.445,395.442,170.750,41.367,157.855
C06159=1038.406,208.196,395.468,170.748,41.366,157.854
C06160=1038.399,207.948,395.494,170.745,41.364,157.854
C06161=1038.392,207.699,395.520,170.743,41.363,157.853
C06162=1038.386,207.451,395.547,170.741,41.361,157.853
C06163=1038.379,207.202,395.574,170.739,41.361,157.853
C06164=1038.372,206.953,395.600,170.736,41.359,157.852
C06165=1038.364,206.638,395.634,170.734,41.357,157.852
C06166=1038.355,206.321,395.667,170.730,41.356,157.851
C06167=1038.347,206.005,395.701,170.728,41.354,157.851
C06168=1038.338,205.689,395.734,170.725,41.352,157.850
C06169=1038.312,204.638,395.841,170.425,41.248,157.812
C06170=1038.306,204.390,395.866,170.421,41.248,157.812
C06171=1038.300,204.141,395.891,170.418,41.247,157.811
C06172=1038.293,203.893,395.916,170.415,41.247,157.811
C06173=1038.286,203.644,395.942,170.413,41.246,157.811
C06174=1038.281,203.395,395.966,170.409,41.245,157.811
C06175=1038.275,203.147,395.991,170.406,41.245,157.810
C06176=1038.269,202.898,396.016,170.403,41.244,157.810
C06177=1038.263,202.649,396.042,170.399,41.243,157.810
C06178=1038.257,202.400,396.066,170.396,41.243,157.809
C06179=1038.250,202.151,396.092,170.394,41.242,157.809
C06180=1038.244,201.903,396.117,170.390,41.241,157.809
C06181=1038.238,201.654,396.142,170.387,41.241,157.809
C06182=1038.233,201.405,396.167,170.384,41.240,157.808
C06183=1038.226,201.157,396.191,170.381,41.240,157.808
C06184=1038.220,200.908,396.217,170.377,41.239,157.808
C06185=1038.214,200.659,396.241,170.374,41.239,157.807
C06186=1038.207,200.410,396.267,170.372,41.238,157.807
C06187=1038.201,200.162,396.291,170.369,41.238,157.807
C06188=1038.195,199.913,396.316,170.365,41.237,157.807
C06189=1038.188,199.665,396.340,170.362,41.237,157.806
C06190=1038.182,199.416,396.365,170.359,41.237,157.806
C06191=1038.175,199.167,396.390,170.356,41.236,157.806
C06192=1038.170,198.918,396.414,170.353,41.236,157.806
C06193=1038.163,198.670,396.439,170.350,41.235,157.805
C06194=1038.157,198.421,396.463,170.347,41.234,157.805
C06195=1038.151,198.173,396.489,170.344,41.234,157.805
C06196=1038.144,197.924,396.513,170.340,41.234,157.805
C06197=1038.138,197.675,396.538,170.337,41.234,157.804
C06198=1038.132,197.426,396.562,170.335,41.233,157.804
C06199=1038.126,197.178,396.587,170.332,41.232,157.804
C06200=1038.119,196.929,396.611,170.328,41.232,157.804
C06201=1038.113,196.680,396.637,170.325,41.232,157.803
C06202=1038.107,196.431,396.661,170.322,41.231,157.803
C06203=1038.101,196.183,396.685,170.319,41.231,157.803
C06204=1038.095,195.934,396.710,170.316,41.230,157.803
C06205=1038.088,195.685,396.734,170.313,41.230,157.802
C06206=1038.082,195.436,396.760,170.310,41.229,157.802
C06207=1038.076,195.188,396.783,170.307,41.229,157.802
C06208=1038.070,194.939,396.808,170.304,41.229,157.802
C06209=1038.063,194.690,396.833,170.301,41.228,157.801
C06210=1038.058,194.442,396.857,170.298,41.227,157.801
C06211=1038.051,194.193,396.881,170.295,41.227,157.801
C06212=1038.045,193.944,396.906,170.292,41.227,157.801
C06213=1038.039,193.696,396.930,170.289,41.227,157.800
C06214=1038.033,193.447,396.954,170.286,41.226,157.800
C06215=1038.026,193.198,396.979,170.283,41.225,157.800
C06216=1038.021,192.950,397.003,170.280,41.225,157.800
C06217=1038.014,192.701,397.027,170.277,41.225,157.799
C06218=1038.008,192.451,397.052,170.274,41.225,157.799
C06219=1038.002,192.204,397.076,170.271,41.224,157.799
C06220=1037.996,191.955,397.101,170.268,41.223,157.799
C06221=1037.990,191.706,397.125,170.265,41.223,157.798
C06222=1037.984,191.457,397.149,170.262,41.223,157.798
C06223=1037.978,191.208,397.174,170.259,41.223,157.798
C06224=1037.972,190.960,397.198,170.256,41.222,157.798
C06225=1037.966,190.711,397.223,170.253,41.221,157.797
C06226=1037.959,190.462,397.247,170.250,41.221,157.797
C06227=1037.954,190.213,397.271,170.247,41.221,157.797
C06228=1037.948,189.964,397.295,170.245,41.220,157.797
C06229=1037.942,189.716,397.320,170.242,41.220,157.796
C06230=1037.932,189.299,397.360,170.236,41.219,157.796
C06231=1037.921,188.883,397.401,170.232,41.219,157.796
C06232=1037.911,188.467,397.441,170.226,41.218,157.795
C06233=1037.901,188.050,397.482,170.222,41.217,157.795
C06234=1037.895,187.801,397.507,170.219,41.217,157.795
C06235=1037.889,187.552,397.531,170.216,41.217,157.794
C06236=1037.884,187.304,397.555,170.213,41.216,157.794
C06237=1037.877,187.055,397.579,170.210,41.216,157.794
C06238=1037.872,186.806,397.603,170.207,41.215,157.794
C06239=1037.865,186.557,397.627,170.205,41.215,157.793
C06240=1037.859,186.309,397.651,170.202,41.215,157.793
C06241=1037.853,186.060,397.675,170.198,41.214,157.793
C06242=1037.847,185.811,397.699,170.196,41.214,157.793
C06243=1037.841,185.562,397.724,170.193,41.214,157.793
C06244=1037.835,185.314,397.747,170.190,41.213,157.792
C06245=1037.830,185.065,397.772,170.187,41.212,157.792
C06246=1037.823,184.816,397.796,170.184,41.212,157.792
C06247=1037.818,184.568,397.820,170.182,41.212,157.792
C06248=1037.811,184.319,397.844,170.179,41.212,157.791
C06249=1037.806,184.070,397.867,170.176,41.211,157.791
C06250=1037.800,183.821,397.891,170.173,41.211,157.791
C06251=1037.794,183.572,397.916,170.170,41.211,157.791
C06252=1037.788,183.323,397.940,170.167,41.210,157.790
C06253=1037.782,183.075,397.963,170.165,41.210,157.790
C06254=1037.775,182.825,397.987,170.162,41.210,157.790
C06255=1037.769,182.577,398.010,170.158,41.210,157.790
C06256=1037.763,182.328,398.034,170.156,41.209,157.790
C06257=1037.756,182.079,398.057,170.153,41.210,157.790
C06258=1037.749,181.830,398.081,170.150,41.209,157.789
C06259=1037.743,181.582,398.104,170.148,41.209,157.789
C06260=1037.737,181.332,398.128,170.145,41.209,157.789
C06261=1037.731,181.084,398.151,170.142,41.209,157.789
C06262=1037.724,180.835,398.175,170.138,41.209,157.789
C06263=1037.719,180.586,398.198,170.136,41.208,157.788
C06264=1037.712,180.337,398.222,170.133,41.208,157.788
C06265=1037.706,180.088,398.245,170.130,41.208,157.788
C06266=1037.700,179.839,398.269,170.128,41.208,157.788
C06267=1037.693,179.591,398.292,170.125,41.208,157.788
C06268=1037.687,179.343,398.315,170.121,41.208,157.787
C06269=1037.680,179.094,398.339,170.119,41.207,157.787
C06270=1037.675,178.845,398.362,170.116,41.208,157.787
C06271=1037.668,178.596,398.386,170.113,41.207,157.787
C06272=1037.662,178.347,398.409,170.111,41.207,157.787
C06273=1037.656,178.098,398.433,170.107,41.207,157.786
C06274=1037.650,177.849,398.456,170.105,41.206,157.786
C06275=1037.643,177.601,398.479,170.102,41.207,157.786
C06276=1037.637,177.351,398.503,170.099,41.206,157.786
C06277=1037.631,177.103,398.526,170.097,41.206,157.786
C06278=1037.622,176.738,398.561,170.093,41.206,157.786
C06279=1037.613,176.372,398.595,170.088,41.206,157.785
C06280=1037.604,176.007,398.629,170.084,41.206,157.785
C06281=1037.595,175.642,398.663,170.080,41.205,157.785
C06282=1037.588,175.392,398.686,170.078,41.205,157.785
C06283=1037.582,175.144,398.710,170.075,41.205,157.784
C06284=1037.577,174.895,398.733,170.072,41.205,157.784
C06285=1037.570,174.645,398.756,170.069,41.205,157.784
C06286=1037.564,174.397,398.780,170.066,41.205,157.784
C06287=1037.558,174.148,398.802,170.064,41.204,157.784
C06288=1037.551,173.900,398.826,170.061,41.205,157.784
C06289=1037.545,173.651,398.849,170.059,41.204,157.783
C06290=1037.539,173.366,398.876,170.056,41.204,157.783
C06291=1037.531,173.081,398.902,170.052,41.204,157.783
C06292=1037.525,172.797,398.929,170.049,41.203,157.783
C06293=1037.517,172.512,398.955,170.046,41.204,157.783
C06294=1037.512,172.263,398.978,170.043,41.204,157.782
C06295=1037.506,172.015,399.002,170.041,41.203,157.782
C06296=1037.499,171.766,399.025,170.038,41.203,157.782
C06297=1037.493,171.517,399.048,170.035,41.203,157.782
C06298=1037.487,171.268,399.071,170.032,41.203,157.782
C06299=1037.481,171.019,399.094,170.029,41.203,157.781
C06300=1037.475,170.770,399.118,170.027,41.203,157.781
C06301=1037.469,170.521,399.141,170.024,41.203,157.781
C06302=1037.463,170.272,399.163,170.022,41.202,157.781
C06303=1037.457,170.023,399.186,170.019,41.203,157.781
C06304=1037.450,169.775,399.210,170.016,41.202,157.781
C06305=1037.445,169.526,399.233,170.013,41.202,157.780
C06306=1037.439,169.277,399.256,170.011,41.202,157.780
C06307=1037.433,169.028,399.279,170.008,41.202,157.780
C06308=1037.427,168.779,399.301,170.006,41.202,157.780
C06309=1037.421,168.531,399.325,170.003,41.201,157.780
C06310=1037.414,168.281,399.348,170.001,41.202,157.780
C06311=1037.408,168.032,399.371,169.997,41.201,157.779
C06312=1037.403,167.784,399.394,169.994,41.201,157.779
C06313=1037.396,167.535,399.416,169.992,41.201,157.779
C06314=1037.391,167.286,399.439,169.989,41.201,157.779
C06315=1037.385,167.037,399.462,169.987,41.201,157.779
C06316=1037.378,166.788,399.486,169.984,41.200,157.779
C06317=1037.373,166.539,399.508,169.982,41.201,157.778
C06318=1037.366,166.291,399.532,169.978,41.200,157.778
C06319=1037.360,166.042,399.554,169.976,41.200,157.778
C06320=1037.355,165.793,399.577,169.973,41.200,157.778
C06321=1037.349,165.544,399.600,169.971,41.200,157.778
C06322=1037.343,165.295,399.623,169.969,41.200,157.778
C06323=1037.337,165.047,399.646,169.966,41.200,157.778
C06324=1037.331,164.798,399.669,169.964,41.200,157.777
C06325=1037.325,164.549,399.692,169.960,41.199,157.777
C06326=1037.319,164.299,399.715,169.958,41.199,157.777
C06327=1037.313,164.050,399.738,169.955,41.199,157.777
C06328=1037.307,163.802,399.760,169.953,41.199,157.777
C06329=1037.301,163.553,399.783,169.950,41.199,157.777
C06330=1037.295,163.304,399.806,169.948,41.199,157.776
C06331=1037.289,163.055,399.829,169.945,41.199,157.776
C06332=1037.283,162.806,399.851,169.942,41.198,157.776
C06333=1037.277,162.558,399.874,169.939,41.199,157.776
C06334=1037.272,162.308,399.897,169.937,41.198,157.776
C06335=1037.266,162.059,399.919,169.935,41.198,157.775
C06336=1037.260,161.810,399.942,169.932,41.198,157.775
C06337=1037.254,161.562,399.965,169.930,41.198,157.775
C06338=1037.248,161.313,399.988,169.926,41.197,157.775
C06339=1037.242,161.064,400.011,169.924,41.198,157.775
C06340=1037.237,160.815,400.034,169.921,41.197,157.775
C06341=1037.230,160.566,400.056,169.919,41.197,157.774
C06342=1037.224,160.317,400.079,169.917,41.197,157.774
C06343=1037.219,160.068,400.101,169.914,41.197,157.774
C06344=1037.213,159.819,400.123,169.912,41.197,157.774
C06345=1037.207,159.570,400.146,169.909,41.197,157.774
C06346=1037.200,159.322,400.169,169.907,41.197,157.774
C06347=1037.194,159.073,400.190,169.903,41.197,157.774
C06348=1037.188,158.824,400.213,169.901,41.197,157.774
C06349=1037.182,158.575,400.236,169.898,41.197,157.773
C06350=1037.177,158.326,400.258,169.896,41.197,157.773
C06351=1037.170,158.077,400.280,169.893,41.197,157.773
C06352=1037.164,157.828,400.303,169.891,41.197,157.773
C06353=1037.158,157.579,400.325,169.888,41.198,157.773
C06354=1037.151,157.294,400.351,169.886,41.197,157.773
C06355=1037.144,157.009,400.376,169.883,41.197,157.772
C06356=1037.137,156.724,400.402,169.879,41.197,157.772
C06357=1037.130,156.438,400.427,169.876,41.197,157.772
C06358=1037.124,156.190,400.449,169.874,41.197,157.772
C06359=1037.117,155.941,400.472,169.871,41.198,157.772
C06360=1037.112,155.692,400.494,169.869,41.197,157.772
C06361=1037.105,155.443,400.516,169.866,41.198,157.772
C06362=1037.099,155.194,400.538,169.864,41.197,157.772
C06363=1037.093,154.945,400.561,169.862,41.198,157.771
C06364=1037.087,154.696,400.582,169.859,41.197,157.771
C06365=1037.081,154.447,400.605,169.857,41.198,157.771
C06366=1037.075,154.198,400.627,169.854,41.198,157.771
C06367=1037.069,153.949,400.649,169.851,41.198,157.771
C06368=1037.063,153.700,400.671,169.848,41.198,157.771
C06369=1037.056,153.451,400.693,169.846,41.198,157.771
C06370=1037.051,153.202,400.716,169.844,41.198,157.771
C06371=1037.044,152.953,400.738,169.841,41.198,157.770
C06372=1037.038,152.704,400.760,169.839,41.198,157.770
C06373=1037.032,152.456,400.782,169.836,41.198,157.770
C06374=1037.026,152.206,400.804,169.834,41.198,157.770
C06375=1037.020,151.957,400.826,169.831,41.198,157.770
C06376=1037.014,151.708,400.848,169.829,41.198,157.770
C06377=1037.008,151.460,400.869,169.826,41.198,157.770
C06378=1037.002,151.211,400.892,169.823,41.198,157.770
C06379=1036.995,150.962,400.913,169.821,41.199,157.769
C06380=1036.990,150.712,400.936,169.818,41.198,157.769
C06381=1036.984,150.464,400.958,169.816,41.199,157.769
C06382=1036.977,150.215,400.980,169.814,41.199,157.769
C06383=1036.971,149.966,401.002,169.811,41.199,157.769
C06384=1036.965,149.717,401.024,169.809,41.199,157.769
C06385=1036.959,149.468,401.045,169.806,41.199,157.769
C06386=1036.953,149.219,401.068,169.804,41.199,157.769
C06387=1036.947,148.970,401.089,169.802,41.199,157.769
C06388=1036.941,148.721,401.111,169.798,41.199,157.768
C06389=1036.935,148.472,401.133,169.796,41.199,157.768
C06390=1036.928,148.223,401.155,169.794,41.199,157.768
C06391=1036.922,147.974,401.177,169.791,41.199,157.768
C06392=1036.916,147.725,401.198,169.789,41.199,157.768
C06393=1036.911,147.476,401.220,169.786,41.200,157.768
C06394=1036.904,147.228,401.242,169.784,41.200,157.768
C06395=1036.898,146.979,401.264,169.782,41.199,157.768
C06396=1036.893,146.729,401.286,169.779,41.200,157.767
C06397=1036.886,146.480,401.307,169.777,41.200,157.767
C06398=1036.879,146.231,401.328,169.774,41.200,157.767
C06399=1036.873,145.982,401.351,169.772,41.200,157.767
C06400=1036.867,145.734,401.372,169.770,41.200,157.767
C06401=1036.861,145.485,401.394,169.767,41.201,157.767
C06402=1036.855,145.235,401.415,169.764,41.200,157.767
C06403=1036.849,144.986,401.437,169.761,41.201,157.767
C06404=1036.843,144.737,401.459,169.759,41.201,157.767
C06405=1036.837,144.488,401.480,169.757,41.201,157.767
C06406=1036.831,144.239,401.502,169.754,41.201,157.766
C06407=1036.825,143.991,401.524,169.752,41.201,157.766
C06408=1036.818,143.741,401.546,169.750,41.201,157.766
C06409=1036.812,143.492,401.567,169.747,41.202,157.766
C06410=1036.805,143.243,401.588,169.745,41.202,157.766
C06411=1036.800,142.995,401.609,169.742,41.202,157.766
C06412=1036.794,142.746,401.631,169.740,41.202,157.766
C06413=1036.787,142.496,401.653,169.738,41.202,157.766
C06414=1036.781,142.247,401.674,169.735,41.203,157.766
C06415=1036.776,141.999,401.696,169.732,41.202,157.765
C06416=1036.770,141.750,401.717,169.730,41.202,157.765
C06417=1036.763,141.500,401.739,169.727,41.203,157.765
C06418=1036.756,141.216,401.763,169.725,41.203,157.765
C06419=1036.749,140.929,401.788,169.722,41.203,157.765
C06420=1036.743,140.644,401.813,169.719,41.203,157.765
C06421=1036.736,140.359,401.837,169.717,41.203,157.765
C06422=1036.730,140.109,401.858,169.714,41.203,157.765
C06423=1036.723,139.860,401.880,169.712,41.203,157.765
C06424=1036.717,139.611,401.901,169.710,41.204,157.764
C06425=1036.712,139.363,401.923,169.707,41.204,157.764
C06426=1036.705,139.113,401.944,169.705,41.204,157.764
C06427=1036.699,138.864,401.965,169.703,41.204,157.764
C06428=1036.692,138.615,401.987,169.700,41.204,157.764
C06429=1036.687,138.367,402.008,169.698,41.205,157.764
C06430=1036.681,138.118,402.030,169.696,41.205,157.764
C06431=1036.674,137.868,402.050,169.693,41.205,157.764
C06432=1036.669,137.620,402.072,169.690,41.205,157.764
C06433=1036.662,137.370,402.093,169.688,41.205,157.764
C06434=1036.656,137.121,402.115,169.685,41.205,157.764
C06435=1036.650,136.873,402.135,169.683,41.206,157.763
C06436=1036.644,136.624,402.157,169.681,41.206,157.763
C06437=1036.638,136.374,402.178,169.678,41.206,157.763
C06438=1036.631,136.125,402.199,169.676,41.206,157.763
C06439=1036.625,135.877,402.220,169.674,41.206,157.763
C06440=1036.619,135.627,402.242,169.671,41.206,157.763
C06441=1036.613,135.378,402.262,169.669,41.207,157.763
C06442=1036.607,135.129,402.284,169.667,41.207,157.763
C06443=1036.601,134.880,402.305,169.664,41.207,157.763
C06444=1036.594,134.631,402.326,169.662,41.208,157.763
C06445=1036.589,134.382,402.347,169.660,41.208,157.763
C06446=1036.583,134.133,402.368,169.657,41.208,157.762
C06447=1036.576,133.884,402.389,169.655,41.208,157.762
C06448=1036.570,133.635,402.410,169.653,41.208,157.762
C06449=1036.564,133.386,402.431,169.650,41.208,157.762
C06450=1036.557,133.137,402.453,169.647,41.209,157.762
C06451=1036.552,132.888,402.473,169.645,41.209,157.762
C06452=1036.545,132.639,402.494,169.642,41.209,157.762
C06453=1036.540,132.390,402.516,169.640,41.209,157.762
C06454=1036.534,132.140,402.536,169.638,41.209,157.762
C06455=1036.527,131.891,402.558,169.636,41.209,157.762
C06456=1036.521,131.643,402.579,169.633,41.210,157.762
C06457=1036.515,131.393,402.600,169.631,41.210,157.762
C06458=1036.509,131.145,402.620,169.629,41.210,157.761
C06459=1036.503,130.895,402.641,169.626,41.211,157.761
C06460=1036.496,130.646,402.662,169.624,41.211,157.761
C06461=1036.490,130.397,402.682,169.622,41.211,157.761
C06462=1036.484,130.148,402.704,169.619,41.212,157.761
C06463=1036.478,129.899,402.724,169.617,41.212,157.761
C06464=1036.471,129.651,402.745,169.615,41.212,157.761
C06465=1036.466,129.401,402.766,169.612,41.212,157.761
C06466=1036.459,129.153,402.787,169.610,41.213,157.761
C06467=1036.453,128.903,402.807,169.608,41.213,157.761
C06468=1036.446,128.654,402.828,169.605,41.213,157.761
C06469=1036.440,128.405,402.848,169.603,41.213,157.761
C06470=1036.434,128.156,402.869,169.601,41.214,157.761
C06471=1036.428,127.906,402.890,169.599,41.214,157.761
C06472=1036.422,127.657,402.910,169.596,41.214,157.760
C06473=1036.415,127.409,402.931,169.594,41.215,157.760
C06474=1036.410,127.159,402.952,169.592,41.215,157.760
C06475=1036.403,126.911,402.973,169.589,41.215,157.760
C06476=1036.397,126.662,402.993,169.587,41.215,157.760
C06477=1036.391,126.412,403.014,169.585,41.216,157.760
C06478=1036.384,126.163,403.035,169.582,41.216,157.760
C06479=1036.378,125.914,403.055,169.580,41.216,157.760
C06480=1036.372,125.665,403.077,169.578,41.217,157.760
C06481=1036.366,125.416,403.096,169.575,41.217,157.760
C06482=1036.359,125.131,403.120,169.572,41.217,157.760
C06483=1036.351,124.845,403.144,169.569,41.218,157.760
C06484=1036.344,124.559,403.167,169.567,41.218,157.760
C06485=1036.337,124.273,403.191,169.564,41.218,157.760
C06486=1036.331,124.024,403.211,169.562,41.218,157.759
C06487=1036.325,123.776,403.232,169.559,41.219,157.759
C06488=1036.319,123.526,403.253,169.557,41.219,157.759
C06489=1036.313,123.277,403.273,169.555,41.219,157.759
C06490=1036.306,123.028,403.294,169.553,41.220,157.759
C06491=1036.300,122.779,403.314,169.550,41.220,157.759
C06492=1036.294,122.529,403.335,169.548,41.220,157.759
C06493=1036.288,122.281,403.354,169.546,41.220,157.759
C06494=1036.281,122.032,403.376,169.544,41.221,157.759
C06495=1036.276,121.783,403.396,169.541,41.221,157.759
C06496=1036.270,121.534,403.416,169.539,41.221,157.759
C06497=1036.263,121.284,403.436,169.537,41.222,157.759
C06498=1036.257,121.036,403.457,169.535,41.222,157.759
C06499=1036.251,120.786,403.478,169.532,41.222,157.759
C06500=1036.245,120.537,403.498,169.530,41.222,157.758
C06501=1036.238,120.288,403.518,169.528,41.222,157.758
C06502=1036.232,120.039,403.538,169.526,41.222,157.758
C06503=1036.226,119.790,403.560,169.523,41.223,157.758
C06504=1036.220,119.541,403.580,169.521,41.223,157.758
C06505=1036.214,119.292,403.600,169.519,41.223,157.758
C06506=1036.208,119.042,403.621,169.517,41.223,157.758
C06507=1036.202,118.794,403.641,169.514,41.224,157.758
C06508=1036.196,118.544,403.661,169.512,41.224,157.758
C06509=1036.190,118.295,403.681,169.510,41.224,157.758
C06510=1036.184,118.047,403.702,169.508,41.225,157.758
C06511=1036.178,117.797,403.723,169.504,41.225,157.758
C06512=1036.172,117.548,403.742,169.502,41.225,157.758
C06513=1036.165,117.299,403.763,169.500,41.225,157.757
C06514=1036.160,117.050,403.783,169.498,41.226,157.757
C06515=1036.154,116.801,403.803,169.496,41.226,157.757
C06516=1036.147,116.551,403.824,169.493,41.226,157.757
C06517=1036.141,116.303,403.844,169.491,41.227,157.757
C06518=1036.136,116.054,403.864,169.489,41.227,157.757
C06519=1036.129,115.804,403.884,169.487,41.227,157.757
C06520=1036.123,115.555,403.904,169.484,41.227,157.757
C06521=1036.117,115.306,403.925,169.482,41.228,157.757
C06522=1036.111,115.057,403.946,169.480,41.228,157.757
C06523=1036.105,114.808,403.966,169.478,41.228,157.757
C06524=1036.099,114.559,403.986,169.476,41.228,157.757
C06525=1036.093,114.310,404.006,169.473,41.228,157.756
C06526=1036.087,114.061,404.027,169.471,41.228,157.756
C06527=1036.081,113.811,404.047,169.469,41.229,157.756
C06528=1036.075,113.563,404.067,169.467,41.229,157.756
C06529=1036.069,113.314,404.087,169.465,41.229,157.756
C06530=1036.063,113.064,404.106,169.462,41.229,157.756
C06531=1036.057,112.815,404.127,169.460,41.230,157.756
C06532=1036.051,112.566,404.147,169.458,41.230,157.756
C06533=1036.044,112.316,404.167,169.456,41.230,157.756
C06534=1036.038,112.068,404.187,169.453,41.231,157.756
C06535=1036.032,111.819,404.207,169.451,41.231,157.756
C06536=1036.025,111.569,404.227,169.449,41.232,157.756
C06537=1036.019,111.321,404.247,169.447,41.232,157.756
C06538=1036.014,111.071,404.266,169.445,41.232,157.756
C06539=1036.007,110.822,404.287,169.442,41.233,157.756
C06540=1036.001,110.573,404.307,169.440,41.233,157.756
C06541=1035.995,110.324,404.327,169.438,41.233,157.756
C06542=1035.989,110.074,404.347,169.436,41.233,157.755
C06543=1035.983,109.825,404.366,169.433,41.234,157.755
C06544=1035.977,109.576,404.386,169.431,41.234,157.755
C06545=1035.970,109.327,404.406,169.429,41.235,157.755
C06546=1035.963,109.041,404.429,169.426,41.235,157.755
C06547=1035.955,108.755,404.451,169.424,41.235,157.755
C06548=1035.949,108.469,404.474,169.421,41.236,157.755
C06549=1035.941,108.184,404.496,169.419,41.236,157.755
C06550=1035.935,107.935,404.516,169.416,41.236,157.755
C06551=1035.929,107.686,404.536,169.414,41.237,157.755
C06552=1035.922,107.436,404.555,169.412,41.238,157.755
C06553=1035.916,107.187,404.575,169.410,41.238,157.755
C06554=1035.910,106.938,404.595,169.407,41.238,157.755
C06555=1035.905,106.689,404.615,169.405,41.238,157.755
C06556=1035.898,106.440,404.635,169.403,41.239,157.755
C06557=1035.891,106.191,404.654,169.401,41.239,157.755
C06558=1035.886,105.942,404.673,169.399,41.239,157.755
C06559=1035.880,105.693,404.693,169.395,41.240,157.755
C06560=1035.873,105.443,404.714,169.394,41.241,157.755
C06561=1035.867,105.194,404.733,169.392,41.241,157.755
C06562=1035.861,104.945,404.752,169.390,41.241,157.754
C06563=1035.855,104.697,404.772,169.388,41.241,157.754
C06564=1035.848,104.446,404.792,169.385,41.242,157.754
C06565=1035.842,104.198,404.812,169.382,41.242,157.754
C06566=1035.837,103.948,404.831,169.380,41.242,157.754
C06567=1035.830,103.700,404.850,169.378,41.242,157.754
C06568=1035.824,103.450,404.870,169.375,41.243,157.754
C06569=1035.818,103.201,404.890,169.374,41.244,157.754
C06570=1035.812,102.952,404.910,169.372,41.244,157.754
C06571=1035.806,102.702,404.929,169.369,41.244,157.754
C06572=1035.799,102.454,404.949,169.367,41.244,157.754
C06573=1035.793,102.205,404.968,169.365,41.245,157.754
C06574=1035.787,101.955,404.988,169.362,41.245,157.754
C06575=1035.781,101.706,405.007,169.360,41.245,157.754
C06576=1035.774,101.457,405.027,169.358,41.245,157.754
C06577=1035.769,101.208,405.046,169.356,41.246,157.754
C06578=1035.763,100.959,405.066,169.354,41.246,157.754
C06579=1035.757,100.709,405.085,169.351,41.246,157.753
C06580=1035.750,100.460,405.105,169.349,41.247,157.753
C06581=1035.744,100.211,405.124,169.347,41.248,157.753
C06582=1035.738,99.962,405.144,169.345,41.248,157.753
C06583=1035.732,99.713,405.163,169.343,41.248,157.753
C06584=1035.726,99.464,405.183,169.340,41.248,157.753
C06585=1035.719,99.215,405.201,169.338,41.249,157.753
C06586=1035.713,98.965,405.221,169.336,41.250,157.753
C06587=1035.706,98.716,405.240,169.334,41.250,157.753
C06588=1035.700,98.467,405.260,169.331,41.250,157.753
C06589=1035.694,98.218,405.278,169.329,41.250,157.753
C06590=1035.688,97.969,405.298,169.327,41.251,157.753
C06591=1035.681,97.719,405.317,169.325,41.252,157.753
C06592=1035.675,97.470,405.337,169.323,41.252,157.753
C06593=1035.669,97.221,405.356,169.320,41.252,157.753
C06594=1035.663,96.972,405.375,169.318,41.252,157.753
C06595=1035.657,96.723,405.394,169.316,41.253,157.753
C06596=1035.651,96.474,405.414,169.314,41.254,157.753
C06597=1035.644,96.225,405.432,169.312,41.254,157.753
C06598=1035.638,95.975,405.452,169.309,41.254,157.753
C06599=1035.631,95.726,405.471,169.307,41.254,157.753
C06600=1035.625,95.477,405.491,169.306,41.255,157.753
C06601=1035.619,95.227,405.509,169.303,41.256,157.753
C06602=1035.613,94.978,405.528,169.301,41.256,157.753
C06603=1035.607,94.730,405.548,169.298,41.256,157.752
C06604=1035.601,94.480,405.567,169.296,41.256,157.752
C06605=1035.594,94.231,405.586,169.295,41.257,157.752
C06606=1035.589,93.982,405.605,169.293,41.258,157.752
C06607=1035.582,93.733,405.624,169.291,41.258,157.752
C06608=1035.576,93.484,405.644,169.287,41.258,157.752
C06609=1035.569,93.234,405.663,169.285,41.258,157.752
C06610=1035.562,92.949,405.685,169.283,41.259,157.752
C06611=1035.555,92.662,405.706,169.281,41.260,157.752
C06612=1035.548,92.377,405.729,169.279,41.260,157.752
C06613=1035.541,92.091,405.750,169.275,41.260,157.752
C06614=1035.536,91.842,405.769,169.273,41.261,157.752
C06615=1035.529,91.593,405.788,169.271,41.261,157.752
C06616=1035.524,91.343,405.807,169.269,41.261,157.752
C06617=1035.517,91.095,405.826,169.268,41.262,157.752
C06618=1035.511,90.845,405.846,169.265,41.262,157.752
C06619=1035.504,90.595,405.865,169.262,41.263,157.752
C06620=1035.498,90.346,405.884,169.260,41.263,157.752
C06621=1035.492,90.097,405.902,169.258,41.263,157.752
C06622=1035.486,89.847,405.922,169.256,41.263,157.752
C06623=1035.480,89.598,405.940,169.254,41.264,157.752
C06624=1035.473,89.349,405.959,169.252,41.265,157.751
C06625=1035.467,89.100,405.978,169.249,41.265,157.751
C06626=1035.461,88.851,405.996,169.248,41.266,157.752
C06627=1035.455,88.601,406.016,169.246,41.266,157.751
C06628=1035.448,88.352,406.034,169.243,41.266,157.751
C06629=1035.442,88.103,406.053,169.241,41.267,157.751
C06630=1035.436,87.854,406.072,169.239,41.268,157.751
C06631=1035.429,87.605,406.090,169.237,41.268,157.751
C06632=1035.423,87.356,406.109,169.234,41.268,157.751
C06633=1035.417,87.106,406.128,169.232,41.269,157.751
C06634=1035.411,86.857,406.147,169.230,41.269,157.751
C06635=1035.404,86.608,406.165,169.228,41.270,157.751
C06636=1035.398,86.359,406.184,169.226,41.270,157.751
C06637=1035.391,86.110,406.203,169.223,41.271,157.751
C06638=1035.386,85.861,406.222,169.221,41.271,157.751
C06639=1035.379,85.611,406.241,169.219,41.271,157.751
C06640=1035.373,85.362,406.259,169.217,41.272,157.751
C06641=1035.366,85.113,406.278,169.215,41.272,157.751
C06642=1035.360,84.864,406.296,169.212,41.273,157.751
C06643=1035.354,84.614,406.314,169.210,41.273,157.751
C06644=1035.348,84.365,406.334,169.208,41.274,157.751
C06645=1035.342,84.116,406.352,169.206,41.274,157.751
C06646=1035.335,83.867,406.371,169.204,41.275,157.751
C06647=1035.329,83.617,406.390,169.202,41.275,157.751
C06648=1035.322,83.368,406.408,169.199,41.276,157.751
C06649=1035.317,83.119,406.427,169.197,41.276,157.751
C06650=1035.311,82.869,406.445,169.195,41.276,157.751
C06651=1035.304,82.620,406.464,169.193,41.277,157.751
C06652=1035.298,82.371,406.483,169.191,41.277,157.751
C06653=1035.292,82.123,406.501,169.188,41.278,157.751
C06654=1035.286,81.873,406.520,169.186,41.278,157.750
C06655=1035.279,81.624,406.538,169.184,41.278,157.750
C06656=1035.274,81.374,406.557,169.182,41.279,157.750
C06657=1035.267,81.125,406.575,169.180,41.279,157.750
C06658=1035.261,80.876,406.594,169.178,41.280,157.750
C06659=1035.254,80.627,406.613,169.175,41.280,157.750
C06660=1035.248,80.378,406.631,169.173,41.280,157.750
C06661=1035.242,80.128,406.649,169.171,41.281,157.750
C06662=1035.236,79.879,406.669,169.169,41.281,157.750
C06663=1035.230,79.630,406.687,169.167,41.282,157.750
C06664=1035.224,79.381,406.706,169.164,41.282,157.750
C06665=1035.218,79.131,406.723,169.162,41.282,157.750
C06666=1035.211,78.882,406.742,169.160,41.283,157.750
C06667=1035.205,78.633,406.761,169.158,41.283,157.750
C06668=1035.199,78.383,406.779,169.156,41.284,157.750
C06669=1035.193,78.134,406.798,169.154,41.284,157.750
C06670=1035.187,77.885,406.817,169.151,41.285,157.750
C06671=1035.181,77.636,406.834,169.149,41.285,157.750
C06672=1035.175,77.387,406.853,169.147,41.286,157.750
C06673=1035.168,77.137,406.871,169.145,41.286,157.750
C06674=1035.161,76.851,406.892,169.142,41.287,157.750
C06675=1035.154,76.566,406.912,169.140,41.287,157.750
C06676=1035.146,76.279,406.934,169.137,41.287,157.750
C06677=1035.139,75.994,406.955,169.135,41.288,157.750
C06678=1035.133,75.745,406.973,169.133,41.289,157.750
C06679=1035.127,75.495,406.991,169.130,41.290,157.750
C06680=1035.120,75.246,407.010,169.128,41.290,157.750
C06681=1035.115,74.997,407.028,169.126,41.290,157.750
C06682=1035.108,74.748,407.046,169.125,41.291,157.750
C06683=1035.101,74.498,407.064,169.123,41.291,157.750
C06684=1035.095,74.249,407.082,169.119,41.292,157.749
C06685=1035.089,73.999,407.100,169.117,41.292,157.749
C06686=1035.082,73.750,407.119,169.116,41.293,157.749
C06687=1035.077,73.501,407.136,169.114,41.293,157.749
C06688=1035.070,73.252,407.155,169.112,41.293,157.749
C06689=1035.064,73.002,407.173,169.109,41.294,157.749
C06690=1035.058,72.753,407.192,169.107,41.295,157.749
C06691=1035.051,72.504,407.209,169.105,41.295,157.749
C06692=1035.045,72.255,407.227,169.103,41.296,157.749
C06693=1035.039,72.006,407.245,169.101,41.296,157.749
C06694=1035.033,71.757,407.264,169.099,41.296,157.749
C06695=1035.027,71.507,407.282,169.096,41.297,157.749
C06696=1035.020,71.258,407.300,169.094,41.297,157.749
C06697=1035.015,71.009,407.318,169.092,41.298,157.749
C06698=1035.008,70.759,407.335,169.090,41.298,157.749
C06699=1035.001,70.510,407.354,169.088,41.299,157.749
C06700=1034.995,70.260,407.372,169.085,41.299,157.749
C06701=1034.989,70.012,407.390,169.083,41.299,157.749
C06702=1034.983,69.762,407.408,169.081,41.300,157.749
C06703=1034.977,69.512,407.426,169.079,41.301,157.749
C06704=1034.970,69.264,407.444,169.077,41.301,157.749
C06705=1034.964,69.014,407.462,169.074,41.301,157.749
C06706=1034.958,68.766,407.480,169.072,41.302,157.749
C06707=1034.952,68.516,407.498,169.070,41.302,157.749
C06708=1034.945,68.266,407.516,169.068,41.303,157.749
C06709=1034.939,68.017,407.533,169.066,41.304,157.749
C06710=1034.933,67.768,407.552,169.063,41.304,157.749
C06711=1034.926,67.519,407.569,169.061,41.305,157.749
C06712=1034.920,67.269,407.587,169.059,41.305,157.749
C06713=1034.914,67.020,407.606,169.057,41.305,157.749
C06714=1034.907,66.771,407.623,169.055,41.306,157.749
C06715=1034.901,66.521,407.641,169.052,41.307,157.749
C06716=1034.895,66.272,407.658,169.050,41.307,157.749
C06717=1034.889,66.024,407.676,169.048,41.308,157.749
C06718=1034.883,65.774,407.694,169.046,41.308,157.749
C06719=1034.876,65.524,407.712,169.044,41.308,157.748
C06720=1034.870,65.275,407.729,169.041,41.309,157.748
C06721=1034.864,65.026,407.748,169.039,41.310,157.748
C06722=1034.858,64.776,407.766,169.037,41.310,157.748
C06723=1034.851,64.527,407.783,169.036,41.311,157.748
C06724=1034.845,64.278,407.800,169.034,41.311,157.748
C06725=1034.838,64.029,407.818,169.030,41.311,157.748
C06726=1034.832,63.779,407.836,169.029,41.312,157.748
C06727=1034.826,63.530,407.854,169.027,41.312,157.748
C06728=1034.820,63.281,407.871,169.025,41.313,157.748
C06729=1034.813,63.032,407.889,169.022,41.314,157.748
C06730=1034.807,62.782,407.907,169.020,41.315,157.748
C06731=1034.800,62.533,407.924,169.018,41.315,157.748
C06732=1034.794,62.284,407.941,169.016,41.316,157.748
C06733=1034.787,62.034,407.959,169.013,41.316,157.748
C06734=1034.781,61.784,407.976,169.011,41.317,157.748
C06735=1034.775,61.535,407.994,169.009,41.317,157.748
C06736=1034.768,61.286,408.011,169.007,41.318,157.748
C06737=1034.761,61.037,408.028,169.004,41.319,157.748
C06738=1034.754,60.751,408.048,169.002,41.320,157.748
C06739=1034.747,60.465,408.068,168.999,41.320,157.748
C06740=1034.740,60.178,408.089,168.997,41.321,157.748
C06741=1034.732,59.892,408.108,168.994,41.321,157.748
C06742=1034.726,59.643,408.126,168.992,41.322,157.748
C06743=1034.720,59.394,408.143,168.990,41.322,157.748
C06744=1034.713,59.145,408.160,168.988,41.323,157.748
C06745=1034.707,58.895,408.178,168.986,41.324,157.748
C06746=1034.700,58.646,408.195,168.984,41.325,157.748
C06747=1034.694,58.397,408.213,168.982,41.325,157.748
C06748=1034.688,58.147,408.230,168.980,41.326,157.748
C06749=1034.681,57.898,408.247,168.977,41.326,157.748
C06750=1034.674,57.649,408.265,168.975,41.326,157.748
C06751=1034.669,57.400,408.282,168.973,41.327,157.748
C06752=1034.662,57.150,408.300,168.971,41.327,157.748
C06753=1034.655,56.901,408.317,168.968,41.328,157.748
C06754=1034.650,56.652,408.335,168.966,41.329,157.748
C06755=1034.643,56.402,408.352,168.964,41.330,157.748
C06756=1034.637,56.154,408.369,168.962,41.330,157.748
C06757=1034.631,55.903,408.386,168.959,41.331,157.748
C06758=1034.624,55.654,408.403,168.957,41.331,157.748
C06759=1034.618,55.405,408.420,168.955,41.331,157.748
C06760=1034.611,55.155,408.438,168.953,41.332,157.748
C06761=1034.605,54.907,408.455,168.950,41.333,157.748
C06762=1034.598,54.657,408.473,168.948,41.334,157.748
C06763=1034.592,54.407,408.491,168.946,41.334,157.748
C06764=1034.586,54.158,408.507,168.945,41.335,157.748
C06765=1034.579,53.909,408.524,168.942,41.335,157.748
C06766=1034.574,53.660,408.542,168.939,41.335,157.748
C06767=1034.567,53.410,408.559,168.938,41.336,157.748
C06768=1034.561,53.162,408.576,168.936,41.337,157.748
C06769=1034.555,52.912,408.594,168.934,41.337,157.748
C06770=1034.549,52.662,408.610,168.931,41.338,157.748
C06771=1034.542,52.413,408.628,168.929,41.338,157.748
C06772=1034.536,52.164,408.645,168.927,41.339,157.748
C06773=1034.529,51.915,408.663,168.925,41.339,157.748
C06774=1034.524,51.665,408.679,168.923,41.340,157.748
C06775=1034.517,51.416,408.696,168.920,41.341,157.748
C06776=1034.511,51.167,408.714,168.918,41.341,157.748
C06777=1034.504,50.917,408.731,168.916,41.342,157.748
C06778=1034.498,50.668,408.747,168.914,41.342,157.748
C06779=1034.492,50.418,408.765,168.911,41.342,157.747
C06780=1034.486,50.169,408.782,168.909,41.343,157.748
C06781=1034.479,49.920,408.800,168.907,41.343,157.747
C06782=1034.474,49.670,408.816,168.905,41.344,157.748
C06783=1034.467,49.421,408.834,168.903,41.345,157.747
C06784=1034.461,49.172,408.851,168.900,41.345,157.747
C06785=1034.454,48.922,408.867,168.898,41.346,157.747
C06786=1034.449,48.673,408.885,168.896,41.346,157.747
C06787=1034.442,48.424,408.902,168.894,41.346,157.747
C06788=1034.436,48.174,408.918,168.891,41.347,157.747
C06789=1034.430,47.925,408.936,168.889,41.348,157.747
C06790=1034.424,47.676,408.953,168.887,41.348,157.747
C06791=1034.418,47.427,408.970,168.885,41.349,157.747
C06792=1034.411,47.177,408.987,168.883,41.349,157.747
C06793=1034.405,46.928,409.005,168.880,41.349,157.747
C06794=1034.399,46.678,409.021,168.878,41.350,157.747
C06795=1034.392,46.429,409.038,168.876,41.351,157.747
C06796=1034.387,46.180,409.055,168.874,41.351,157.747
C06797=1034.380,45.930,409.072,168.873,41.352,157.747
C06798=1034.374,45.681,409.089,168.869,41.352,157.747
C06799=1034.368,45.431,409.106,168.867,41.352,157.747
C06800=1034.362,45.182,409.123,168.866,41.353,157.747
C06801=1034.356,44.933,409.140,168.864,41.354,157.747
C06802=1034.348,44.646,409.160,168.861,41.354,157.747
C06803=1034.341,44.360,409.179,168.859,41.355,157.747
C06804=1034.334,44.074,409.199,168.856,41.355,157.747
C06805=1034.327,43.788,409.218,168.854,41.355,157.747
C06806=1034.321,43.538,409.235,168.851,41.356,157.747
C06807=1034.315,43.289,409.252,168.849,41.357,157.747
C06808=1034.309,43.039,409.268,168.847,41.357,157.747
C06809=1034.303,42.790,409.286,168.845,41.358,157.747
C06810=1034.297,42.540,409.302,168.842,41.358,157.747
C06811=1034.290,42.291,409.319,168.840,41.359,157.747
C06812=1034.284,42.042,409.336,168.838,41.359,157.747
C06813=1034.278,41.793,409.352,168.836,41.360,157.747
C06814=1034.271,41.543,409.369,168.833,41.361,157.747
C06815=1034.265,41.294,409.385,168.831,41.362,157.747
C06816=1034.259,41.045,409.402,168.829,41.362,157.747
C06817=1034.252,40.795,409.419,168.827,41.363,157.747
C06818=1034.246,40.546,409.436,168.824,41.363,157.747
C06819=1034.240,40.297,409.452,168.822,41.363,157.747
C06820=1034.233,40.047,409.469,168.820,41.364,157.747
C06821=1034.227,39.798,409.486,168.818,41.365,157.747
C06822=1034.221,39.548,409.502,168.815,41.366,157.747
C06823=1034.215,39.298,409.519,168.813,41.366,157.746
C06824=1034.208,39.050,409.536,168.812,41.367,157.747
C06825=1034.202,38.800,409.552,168.810,41.367,157.746
C06826=1034.196,38.550,409.569,168.806,41.367,157.746
C06827=1034.190,38.302,409.585,168.805,41.368,157.746
C06828=1034.184,38.052,409.602,168.803,41.369,157.746
C06829=1034.177,37.802,409.618,168.801,41.369,157.746
C06830=1034.171,37.554,409.635,168.798,41.370,157.746
C06831=1034.165,37.304,409.652,168.796,41.370,157.746
C06832=1034.158,37.054,409.668,168.794,41.371,157.746
C06833=1034.152,36.805,409.684,168.792,41.371,157.746
C06834=1034.146,36.556,409.701,168.789,41.372,157.746
C06835=1034.139,36.306,409.717,168.787,41.373,157.746
C06836=1034.133,36.057,409.734,168.785,41.373,157.746
C06837=1034.126,35.808,409.749,168.782,41.374,157.746
C06838=1034.120,35.558,409.766,168.780,41.375,157.746
C06839=1034.114,35.308,409.782,168.778,41.376,157.746
C06840=1034.108,35.060,409.799,168.775,41.376,157.746
C06841=1034.100,34.810,409.815,168.773,41.377,157.746
C06842=1034.094,34.561,409.832,168.771,41.377,157.746
C06843=1034.088,34.311,409.848,168.769,41.378,157.746
C06844=1034.082,34.062,409.864,168.766,41.378,157.746
C06845=1034.075,33.812,409.880,168.765,41.379,157.746
C06846=1034.069,33.563,409.896,168.763,41.380,157.746
C06847=1034.063,33.314,409.913,168.760,41.381,157.746
C06848=1034.057,33.065,409.930,168.758,41.381,157.746
C06849=1034.050,32.815,409.946,168.756,41.382,157.746
C06850=1034.044,32.566,409.962,168.754,41.382,157.746
C06851=1034.038,32.316,409.978,168.751,41.383,157.746
C06852=1034.032,32.067,409.994,168.749,41.383,157.746
C06853=1034.025,31.817,410.010,168.747,41.384,157.746
C06854=1034.019,31.568,410.027,168.744,41.385,157.746
C06855=1034.013,31.319,410.043,168.742,41.386,157.746
C06856=1034.007,31.069,410.059,168.740,41.386,157.746
C06857=1033.999,30.820,410.075,168.737,41.387,157.746
C06858=1033.993,30.570,410.091,168.735,41.387,157.746
C06859=1033.987,30.321,410.108,168.733,41.388,157.746
C06860=1033.982,30.071,410.124,168.731,41.388,157.746
C06861=1033.975,29.822,410.140,168.728,41.389,157.746
C06862=1033.968,29.572,410.156,168.726,41.390,157.746
C06863=1033.962,29.323,410.172,168.725,41.390,157.746
C06864=1033.956,29.074,410.189,168.721,41.391,157.746
C06865=1033.950,28.825,410.204,168.720,41.392,157.746
C06866=1033.942,28.538,410.223,168.718,41.392,157.746
C06867=1033.936,28.252,410.242,168.715,41.393,157.746
C06868=1033.929,27.965,410.260,168.712,41.393,157.746
C06869=1033.921,27.679,410.279,168.710,41.394,157.746
C06870=1033.914,27.430,410.295,168.707,41.395,157.746
C06871=1033.909,27.180,410.311,168.705,41.396,157.746
C06872=1033.901,26.931,410.327,168.703,41.397,157.746
C06873=1033.895,26.681,410.343,168.700,41.397,157.746
C06874=1033.889,26.432,410.359,168.698,41.398,157.746
C06875=1033.883,26.182,410.374,168.696,41.398,157.746
C06876=1033.877,25.933,410.391,168.693,41.399,157.746
C06877=1033.870,25.684,410.406,168.691,41.399,157.746
C06878=1033.864,25.434,410.423,168.689,41.400,157.746
C06879=1033.857,25.185,410.438,168.686,41.401,157.746
C06880=1033.851,24.935,410.455,168.684,41.402,157.746
C06881=1033.845,24.686,410.470,168.683,41.402,157.746
C06882=1033.839,24.436,410.486,168.680,41.403,157.746
C06883=1033.832,24.187,410.502,168.678,41.404,157.746
C06884=1033.826,23.938,410.518,168.676,41.404,157.746
C06885=1033.819,23.688,410.534,168.673,41.405,157.746
C06886=1033.813,23.438,410.549,168.671,41.405,157.746
C06887=1033.807,23.189,410.565,168.669,41.406,157.746
C06888=1033.801,22.940,410.581,168.666,41.407,157.746
C06889=1033.794,22.691,410.597,168.664,41.407,157.746
C06890=1033.788,22.441,410.613,168.662,41.408,157.746
C06891=1033.782,22.192,410.628,168.659,41.409,157.746
C06892=1033.775,21.943,410.644,168.657,41.410,157.746
C06893=1033.769,21.694,410.660,168.655,41.410,157.746
C06894=1033.763,21.444,410.675,168.652,41.411,157.746
C06895=1033.756,21.194,410.692,168.650,41.411,157.746
C06896=1033.749,20.945,410.707,168.648,41.412,157.746
C06897=1033.744,20.695,410.723,168.645,41.413,157.746
C06898=1033.737,20.446,410.739,168.644,41.413,157.746
C06899=1033.731,20.196,410.755,168.642,41.414,157.746
C06900=1033.725,19.947,410.770,168.639,41.415,157.746
C06901=1033.719,19.697,410.786,168.637,41.416,157.746
C06902=1033.712,19.448,410.802,168.635,41.416,157.746
C06903=1033.706,19.199,410.817,168.632,41.417,157.746
C06904=1033.700,18.949,410.833,168.630,41.417,157.746
C06905=1033.693,18.700,410.848,168.628,41.418,157.746
C06906=1033.687,18.450,410.864,168.625,41.419,157.746
C06907=1033.681,18.201,410.880,168.623,41.419,157.746
C06908=1033.674,17.952,410.895,168.620,41.420,157.746
C06909=1033.668,17.702,410.911,168.618,41.421,157.746
C06910=1033.662,17.453,410.926,168.616,41.422,157.746
C06911=1033.655,17.204,410.942,168.613,41.423,157.746
C06912=1033.650,16.954,410.957,168.611,41.423,157.746
C06913=1033.643,16.705,410.973,168.610,41.424,157.746
C06914=1033.636,16.455,410.988,168.607,41.424,157.746
C06915=1033.631,16.206,411.004,168.605,41.425,157.746
C06916=1033.624,15.957,411.020,168.603,41.425,157.746
C06917=1033.617,15.707,411.035,168.600,41.426,157.746
C06918=1033.611,15.458,411.050,168.598,41.427,157.746
C06919=1033.605,15.208,411.066,168.595,41.428,157.746
C06920=1033.599,14.958,411.081,168.593,41.429,157.746
C06921=1033.592,14.709,411.096,168.591,41.429,157.746
C06922=1033.586,14.459,411.112,168.588,41.430,157.746
C06923=1033.580,14.210,411.128,168.586,41.430,157.746
C06924=1033.573,13.961,411.143,168.584,41.431,157.746
C06925=1033.567,13.711,411.159,168.581,41.432,157.746
C06926=1033.561,13.462,411.174,168.579,41.432,157.746
C06927=1033.555,13.212,411.189,168.576,41.433,157.746
C06928=1033.548,12.963,411.204,168.575,41.434,157.746
C06929=1033.542,12.713,411.219,168.573,41.435,157.746
C06930=1033.534,12.428,411.237,168.570,41.436,157.746
C06931=1033.526,12.143,411.255,168.567,41.437,157.746
C06932=1033.519,11.857,411.272,168.564,41.438,157.746
C06933=1033.512,11.572,411.289,168.562,41.439,157.746
C06934=1033.506,11.323,411.304,168.559,41.439,157.746
C06935=1033.499,11.074,411.320,168.557,41.440,157.746
C06936=1033.493,10.824,411.334,168.554,41.441,157.746
C06937=1033.486,10.574,411.349,168.552,41.442,157.746
C06938=1033.480,10.325,411.365,168.549,41.442,157.746
C06939=1033.473,10.076,411.380,168.548,41.443,157.746
C06940=1033.467,9.826,411.395,168.546,41.444,157.746
C06941=1033.461,9.576,411.410,168.543,41.444,157.746
C06942=1033.454,9.327,411.426,168.541,41.445,157.746
C06943=1033.448,9.078,411.441,168.538,41.446,157.746
C06944=1033.441,8.828,411.455,168.536,41.447,157.746
C06945=1033.435,8.578,411.470,168.533,41.448,157.746
C06946=1033.429,8.330,411.486,168.531,41.449,157.746
C06947=1033.422,8.080,411.501,168.529,41.449,157.746
C06948=1033.416,7.831,411.516,168.526,41.450,157.746
C06949=1033.410,7.581,411.531,168.524,41.451,157.746
C06950=1033.404,7.331,411.546,168.521,41.451,157.746
C06951=1033.397,7.082,411.562,168.519,41.452,157.746
C06952=1033.391,6.832,411.577,168.518,41.453,157.746
C06953=1033.384,6.583,411.592,168.515,41.453,157.746
C06954=1033.379,6.334,411.606,168.513,41.454,157.746
C06955=1033.372,6.084,411.621,168.510,41.455,157.746
C06956=1033.366,5.835,411.636,168.508,41.456,157.746
C06957=1033.359,5.585,411.652,168.505,41.457,157.746
C06958=1033.353,5.336,411.667,168.503,41.458,157.746
C06959=1033.346,5.086,411.682,168.501,41.458,157.746
C06960=1033.340,4.837,411.697,168.498,41.459,157.746
C06961=1033.334,4.588,411.711,168.496,41.460,157.746
C06962=1033.328,4.338,411.726,168.493,41.460,157.746
C06963=1033.322,4.088,411.741,168.491,41.461,157.746
C06964=1033.315,3.839,411.756,168.489,41.462,157.746
C06965=1033.309,3.589,411.771,168.486,41.462,157.746
C06966=1033.303,3.340,411.786,168.485,41.463,157.746
C06967=1033.296,3.091,411.801,168.482,41.464,157.746
C06968=1033.290,2.841,411.816,168.480,41.465,157.746
C06969=1033.284,2.592,411.831,168.477,41.466,157.746
C06970=1033.277,2.342,411.846,168.475,41.466,157.746
C06971=1033.271,2.093,411.861,168.472,41.467,157.746
C06972=1033.265,1.843,411.876,168.470,41.468,157.746
C06973=1033.259,1.594,411.891,168.467,41.468,157.746
C06974=1033.252,1.344,411.905,168.465,41.469,157.746
C06975=1033.246,1.095,411.920,168.463,41.469,157.746
C06976=1033.240,0.845,411.935,168.460,41.470,157.746
C06977=1033.234,0.596,411.950,168.458,41.471,157.746
C06978=1033.227,0.346,411.965,168.455,41.472,157.746
C06979=1033.221,0.097,411.979,168.454,41.473,157.746
C06980=1033.215,-0.153,411.994,168.450,41.473,157.746
C06981=1033.209,-0.402,412.009,168.449,41.474,157.746
C06982=1033.202,-0.652,412.024,168.447,41.475,157.746
C06983=1033.197,-0.901,412.039,168.444,41.475,157.746
C06984=1033.190,-1.150,412.054,168.442,41.476,157.746
C06985=1033.184,-1.401,412.068,168.439,41.477,157.746
C06986=1033.178,-1.650,412.083,168.437,41.477,157.746
C06987=1033.172,-1.899,412.098,168.434,41.479,157.746
C06988=1033.166,-2.149,412.113,168.432,41.479,157.746
C06989=1033.160,-2.398,412.127,168.430,41.480,157.746
C06990=1033.153,-2.648,412.142,168.427,41.480,157.746
C06991=1033.147,-2.897,412.157,168.425,41.481,157.746
C06992=1033.141,-3.146,412.172,168.422,41.482,157.746
C06993=1033.135,-3.396,412.187,168.420,41.482,157.746
C06994=1033.128,-3.679,412.203,168.418,41.483,157.746
C06995=1033.121,-3.963,412.219,168.415,41.484,157.746
C06996=1033.113,-4.246,412.236,168.412,41.485,157.746
C06997=1033.105,-4.529,412.252,168.409,41.486,157.746
C06998=1033.099,-4.778,412.267,168.407,41.487,157.746
C06999=1033.094,-5.028,412.281,168.404,41.488,157.746
C07000=1033.086,-5.277,412.295,168.402,41.489,157.746
C07001=1033.080,-5.527,412.310,168.399,41.490,157.746
C07002=1033.075,-5.777,412.324,168.397,41.490,157.746
C07003=1033.068,-6.026,412.338,168.394,41.491,157.746
C07004=1033.061,-6.276,412.353,168.392,41.492,157.746
C07005=1033.056,-6.525,412.367,168.390,41.493,157.746
C07006=1033.049,-6.775,412.382,168.388,41.494,157.746
C07007=1033.042,-7.024,412.396,168.385,41.494,157.746
C07008=1033.036,-7.273,412.410,168.383,41.495,157.746
C07009=1033.030,-7.523,412.425,168.380,41.496,157.746
C07010=1033.023,-7.773,412.440,168.378,41.497,157.746
C07011=1033.017,-8.022,412.453,168.375,41.498,157.746
C07012=1033.011,-8.272,412.468,168.373,41.498,157.746
C07013=1033.004,-8.521,412.483,168.370,41.500,157.746
C07014=1032.998,-8.771,412.496,168.368,41.500,157.746
C07015=1032.992,-9.020,412.511,168.365,41.501,157.746
C07016=1032.986,-9.269,412.526,168.364,41.502,157.746
C07017=1032.979,-9.519,412.539,168.361,41.503,157.746
C07018=1032.973,-9.769,412.554,168.359,41.504,157.746
C07019=1032.966,-10.018,412.567,168.356,41.505,157.746
C07020=1032.960,-10.268,412.582,168.354,41.505,157.746
C07021=1032.955,-10.517,412.596,168.351,41.506,157.746
C07022=1032.947,-10.767,412.611,168.349,41.507,157.746
C07023=1032.942,-11.016,412.624,168.346,41.508,157.746
C07024=1032.935,-11.266,412.639,168.343,41.508,157.746
C07025=1032.928,-11.515,412.654,168.341,41.509,157.746
C07026=1032.923,-11.765,412.668,168.339,41.510,157.746
C07027=1032.916,-12.014,412.682,168.336,41.511,157.746
C07028=1032.910,-12.264,412.696,168.334,41.512,157.746
C07029=1032.904,-12.513,412.711,168.332,41.513,157.746
C07030=1032.898,-12.763,412.724,168.329,41.514,157.746
C07031=1032.891,-13.012,412.739,168.327,41.514,157.746
C07032=1032.885,-13.262,412.752,168.324,41.515,157.746
C07033=1032.879,-13.511,412.767,168.322,41.516,157.746
C07034=1032.873,-13.761,412.781,168.319,41.517,157.746
C07035=1032.866,-14.011,412.795,168.317,41.517,157.746
C07036=1032.861,-14.260,412.809,168.314,41.518,157.746
C07037=1032.854,-14.510,412.823,168.312,41.519,157.746
C07038=1032.848,-14.759,412.838,168.309,41.520,157.746
C07039=1032.842,-15.009,412.852,168.308,41.520,157.746
C07040=1032.835,-15.258,412.866,168.305,41.522,157.746
C07041=1032.829,-15.508,412.880,168.302,41.523,157.746
C07042=1032.823,-15.758,412.894,168.300,41.523,157.746
C07043=1032.816,-16.006,412.908,168.297,41.524,157.746
C07044=1032.810,-16.257,412.922,168.295,41.525,157.746
C07045=1032.804,-16.506,412.935,168.292,41.526,157.746
C07046=1032.797,-16.755,412.949,168.290,41.527,157.746
C07047=1032.791,-17.005,412.963,168.287,41.528,157.746
C07048=1032.784,-17.255,412.977,168.285,41.529,157.746
C07049=1032.779,-17.505,412.991,168.283,41.530,157.747
C07050=1032.772,-17.754,413.005,168.280,41.531,157.747
C07051=1032.766,-18.003,413.018,168.278,41.531,157.746
C07052=1032.760,-18.253,413.033,168.275,41.532,157.747
C07053=1032.753,-18.503,413.046,168.272,41.533,157.747
C07054=1032.747,-18.751,413.060,168.270,41.534,157.747
C07055=1032.741,-19.002,413.074,168.267,41.535,157.747
C07056=1032.734,-19.251,413.087,168.265,41.536,157.747
C07057=1032.728,-19.501,413.101,168.263,41.537,157.747
C07058=1032.721,-19.782,413.117,168.260,41.538,157.747
C07059=1032.713,-20.064,413.133,168.257,41.539,157.747
C07060=1032.707,-20.345,413.148,168.254,41.540,157.747
C07061=1032.700,-20.627,413.164,168.251,41.541,157.747
C07062=1032.693,-20.877,413.177,168.249,41.542,157.747
C07063=1032.687,-21.126,413.191,168.246,41.543,157.747
C07064=1032.681,-21.376,413.205,168.243,41.544,157.747
C07065=1032.674,-21.625,413.218,168.241,41.545,157.747
C07066=1032.668,-21.875,413.231,168.239,41.546,157.747
C07067=1032.662,-22.124,413.246,168.237,41.547,157.747
C07068=1032.656,-22.374,413.260,168.234,41.547,157.747
C07069=1032.649,-22.624,413.273,168.231,41.548,157.747
C07070=1032.643,-22.873,413.287,168.229,41.549,157.747
C07071=1032.637,-23.122,413.300,168.226,41.550,157.747
C07072=1032.630,-23.372,413.314,168.224,41.551,157.747
C07073=1032.625,-23.622,413.328,168.221,41.552,157.747
C07074=1032.619,-23.871,413.341,168.218,41.552,157.747
C07075=1032.612,-24.121,413.355,168.216,41.553,157.747
C07076=1032.606,-24.370,413.369,168.214,41.554,157.747
C07077=1032.600,-24.619,413.383,168.212,41.555,157.747
C07078=1032.593,-24.869,413.396,168.209,41.556,157.747
C07079=1032.587,-25.119,413.409,168.206,41.557,157.747
C07080=1032.581,-25.368,413.423,168.204,41.558,157.747
C07081=1032.574,-25.618,413.437,168.201,41.559,157.747
C07082=1032.568,-25.867,413.450,168.199,41.560,157.747
C07083=1032.563,-26.117,413.464,168.196,41.561,157.747
C07084=1032.556,-26.367,413.478,168.193,41.562,157.747
C07085=1032.550,-26.616,413.491,168.191,41.562,157.747
C07086=1032.543,-26.865,413.504,168.189,41.563,157.747
C07087=1032.538,-27.115,413.518,168.187,41.564,157.747
C07088=1032.531,-27.365,413.532,168.184,41.565,157.747
C07089=1032.525,-27.615,413.544,168.181,41.566,157.747
C07090=1032.519,-27.864,413.558,168.179,41.567,157.747
C07091=1032.512,-28.114,413.571,168.176,41.568,157.747
C07092=1032.506,-28.363,413.585,168.173,41.569,157.747
C07093=1032.500,-28.613,413.598,168.171,41.570,157.747
C07094=1032.493,-28.863,413.611,168.169,41.571,157.747
C07095=1032.487,-29.112,413.625,168.166,41.572,157.747
C07096=1032.481,-29.361,413.638,168.164,41.573,157.747
C07097=1032.475,-29.611,413.651,168.161,41.574,157.747
C07098=1032.468,-29.861,413.664,168.158,41.575,157.747
C07099=1032.462,-30.110,413.677,168.155,41.576,157.748
C07100=1032.455,-30.359,413.691,168.153,41.577,157.748
C07101=1032.449,-30.609,413.704,168.150,41.578,157.748
C07102=1032.443,-30.859,413.717,168.148,41.579,157.748
C07103=1032.436,-31.109,413.730,168.146,41.580,157.748
C07104=1032.430,-31.358,413.743,168.143,41.581,157.748
C07105=1032.424,-31.607,413.757,168.140,41.582,157.748
C07106=1032.417,-31.857,413.770,168.138,41.583,157.748
C07107=1032.411,-32.107,413.783,168.135,41.584,157.748
C07108=1032.405,-32.356,413.796,168.132,41.585,157.748
C07109=1032.399,-32.605,413.809,168.130,41.586,157.748
C07110=1032.393,-32.855,413.822,168.127,41.587,157.748
C07111=1032.386,-33.105,413.836,168.125,41.588,157.748
C07112=1032.380,-33.355,413.849,168.123,41.589,157.748
C07113=1032.374,-33.604,413.862,168.120,41.590,157.748
C07114=1032.368,-33.854,413.875,168.117,41.591,157.748
C07115=1032.362,-34.103,413.888,168.115,41.592,157.748
C07116=1032.355,-34.353,413.902,168.112,41.593,157.748
C07117=1032.349,-34.603,413.914,168.109,41.594,157.748
C07118=1032.343,-34.852,413.927,168.107,41.595,157.748
C07119=1032.336,-35.101,413.941,168.105,41.596,157.748
C07120=1032.331,-35.351,413.953,168.102,41.597,157.748
C07121=1032.324,-35.601,413.967,168.099,41.598,157.748
C07122=1032.319,-35.819,413.978,168.097,41.599,157.748
C07123=1032.314,-36.037,413.990,168.095,41.599,157.748
C07124=1032.308,-36.255,414.001,168.092,41.600,157.748
C07125=1032.303,-36.473,414.013,168.090,41.601,157.748
C07126=1032.297,-36.692,414.024,168.088,41.602,157.748
C07127=1032.292,-36.909,414.035,168.085,41.603,157.748
C07128=1032.287,-37.128,414.047,168.083,41.603,157.748
C07129=1032.281,-37.347,414.058,168.082,41.604,157.748
C07130=1032.273,-37.690,414.076,168.078,41.606,157.748
C07131=1032.264,-38.033,414.093,168.074,41.607,157.748
C07132=1032.256,-38.376,414.112,168.071,41.608,157.748
C07133=1032.247,-38.721,414.129,168.067,41.609,157.748
C07134=1032.241,-38.970,414.142,168.064,41.611,157.748
C07135=1032.235,-39.220,414.155,168.061,41.612,157.748
C07136=1032.229,-39.470,414.168,168.060,41.613,157.749
C07137=1032.222,-39.719,414.180,168.057,41.614,157.749
C07138=1032.216,-39.968,414.194,168.054,41.615,157.749
C07139=1032.210,-40.218,414.206,168.051,41.616,157.749
C07140=1032.204,-40.468,414.219,168.049,41.617,157.749
C07141=1032.197,-40.717,414.231,168.046,41.618,157.749
C07142=1032.191,-40.968,414.244,168.044,41.619,157.749
C07143=1032.184,-41.217,414.257,168.041,41.620,157.749
C07144=1032.179,-41.467,414.270,168.039,41.621,157.749
C07145=1032.172,-41.716,414.282,168.036,41.622,157.749
C07146=1032.166,-41.966,414.295,168.033,41.623,157.749
C07147=1032.160,-42.216,414.308,168.030,41.625,157.749
C07148=1032.153,-42.465,414.321,168.028,41.626,157.749
C07149=1032.147,-42.714,414.333,168.026,41.627,157.749
C07150=1032.141,-42.964,414.346,168.023,41.628,157.749
C07151=1032.135,-43.214,414.359,168.020,41.629,157.749
C07152=1032.128,-43.463,414.371,168.018,41.630,157.749
C07153=1032.122,-43.713,414.383,168.015,41.631,157.749
C07154=1032.116,-43.963,414.396,168.012,41.632,157.749
C07155=1032.109,-44.212,414.409,168.009,41.633,157.749
C07156=1032.103,-44.462,414.421,168.006,41.634,157.749
C07157=1032.098,-44.712,414.434,168.005,41.635,157.749
C07158=1032.091,-44.961,414.446,168.002,41.636,157.749
C07159=1032.085,-45.210,414.459,167.999,41.638,157.749
C07160=1032.079,-45.460,414.472,167.996,41.639,157.749
C07161=1032.073,-45.710,414.484,167.994,41.640,157.750
C07162=1032.066,-45.959,414.497,167.991,41.641,157.750
C07163=1032.060,-46.209,414.509,167.989,41.642,157.750
C07164=1032.054,-46.459,414.522,167.986,41.643,157.750
C07165=1032.047,-46.709,414.534,167.984,41.644,157.750
C07166=1032.041,-46.958,414.547,167.981,41.645,157.750
C07167=1032.036,-47.207,414.559,167.978,41.646,157.750
C07168=1032.029,-47.457,414.571,167.975,41.647,157.750
C07169=1032.023,-47.706,414.584,167.972,41.649,157.750
C07170=1032.017,-47.956,414.596,167.970,41.649,157.750
C07171=1032.011,-48.206,414.608,167.968,41.651,157.750
C07172=1032.005,-48.455,414.622,167.965,41.652,157.750
C07173=1031.999,-48.705,414.634,167.962,41.653,157.750
C07174=1031.992,-48.955,414.646,167.960,41.654,157.750
C07175=1031.986,-49.204,414.659,167.957,41.655,157.750
C07176=1031.980,-49.454,414.671,167.954,41.656,157.750
C07177=1031.974,-49.703,414.683,167.951,41.657,157.750
C07178=1031.968,-49.953,414.695,167.950,41.658,157.750
C07179=1031.962,-50.203,414.708,167.947,41.659,157.750
C07180=1031.956,-50.452,414.721,167.944,41.661,157.750
C07181=1031.950,-50.702,414.733,167.941,41.662,157.750
C07182=1031.943,-50.951,414.745,167.938,41.663,157.750
C07183=1031.937,-51.201,414.758,167.935,41.664,157.750
C07184=1031.931,-51.451,414.769,167.934,41.665,157.750
C07185=1031.924,-51.701,414.781,167.931,41.666,157.750
C07186=1031.917,-51.982,414.795,167.927,41.668,157.751
C07187=1031.910,-52.264,414.809,167.924,41.669,157.751
C07188=1031.903,-52.544,414.822,167.921,41.671,157.751
C07189=1031.896,-52.826,414.836,167.919,41.672,157.751
C07190=1031.890,-53.075,414.847,167.916,41.673,157.751
C07191=1031.883,-53.325,414.859,167.913,41.675,157.751
C07192=1031.877,-53.575,414.872,167.910,41.676,157.751
C07193=1031.870,-53.824,414.884,167.907,41.677,157.751
C07194=1031.864,-54.074,414.896,167.904,41.679,157.751
C07195=1031.858,-54.324,414.908,167.903,41.680,157.751
C07196=1031.852,-54.573,414.919,167.900,41.681,157.751
C07197=1031.845,-54.823,414.931,167.897,41.682,157.751
C07198=1031.840,-55.073,414.944,167.894,41.684,157.751
C07199=1031.833,-55.322,414.956,167.891,41.685,157.751
C07200=1031.826,-55.572,414.968,167.888,41.686,157.751
C07201=1031.820,-55.821,414.980,167.886,41.687,157.751
C07202=1031.815,-56.071,414.991,167.883,41.688,157.751
C07203=1031.808,-56.321,415.003,167.881,41.689,157.752
C07204=1031.801,-56.570,415.015,167.878,41.690,157.752
C07205=1031.795,-56.820,415.027,167.875,41.692,157.752
C07206=1031.789,-57.070,415.040,167.872,41.693,157.752
C07207=1031.783,-57.319,415.050,167.870,41.694,157.752
C07208=1031.776,-57.569,415.062,167.867,41.696,157.752
C07209=1031.770,-57.819,415.075,167.864,41.697,157.752
C07210=1031.764,-58.068,415.087,167.861,41.698,157.752
C07211=1031.758,-58.318,415.098,167.859,41.700,157.752
C07212=1031.751,-58.567,415.110,167.857,41.701,157.752
C07213=1031.746,-58.817,415.122,167.854,41.702,157.752
C07214=1031.740,-59.067,415.133,167.851,41.703,157.752
C07215=1031.733,-59.316,415.145,167.848,41.705,157.752
C07216=1031.726,-59.566,415.157,167.845,41.706,157.752
C07217=1031.721,-59.816,415.170,167.842,41.707,157.752
C07218=1031.715,-60.065,415.180,167.840,41.709,157.752
C07219=1031.708,-60.315,415.192,167.838,41.710,157.752
C07220=1031.702,-60.564,415.204,167.835,41.711,157.753
C07221=1031.697,-60.814,415.216,167.832,41.712,157.753
C07222=1031.690,-61.064,415.228,167.829,41.713,157.753
C07223=1031.683,-61.313,415.240,167.826,41.714,157.753
C07224=1031.678,-61.563,415.251,167.824,41.716,157.753
C07225=1031.672,-61.813,415.263,167.821,41.717,157.753
C07226=1031.665,-62.063,415.274,167.818,41.718,157.753
C07227=1031.659,-62.312,415.286,167.815,41.719,157.753
C07228=1031.653,-62.561,415.298,167.813,41.720,157.753
C07229=1031.647,-62.812,415.310,167.811,41.722,157.753
C07230=1031.641,-63.061,415.321,167.808,41.723,157.753
C07231=1031.635,-63.311,415.333,167.805,41.724,157.753
C07232=1031.628,-63.560,415.345,167.802,41.726,157.753
C07233=1031.623,-63.810,415.356,167.799,41.727,157.753
C07234=1031.616,-64.060,415.368,167.796,41.728,157.753
C07235=1031.610,-64.309,415.380,167.793,41.729,157.753
C07236=1031.604,-64.559,415.391,167.791,41.731,157.753
C07237=1031.597,-64.808,415.403,167.789,41.732,157.753
C07238=1031.592,-65.058,415.414,167.786,41.733,157.754
C07239=1031.586,-65.308,415.426,167.783,41.735,157.754
C07240=1031.580,-65.557,415.437,167.780,41.736,157.754
C07241=1031.573,-65.807,415.449,167.778,41.737,157.754
C07242=1031.568,-66.057,415.461,167.775,41.738,157.754
C07243=1031.562,-66.306,415.473,167.772,41.740,157.754
C07244=1031.555,-66.556,415.484,167.769,41.741,157.754
C07245=1031.549,-66.806,415.495,167.766,41.742,157.754
C07246=1031.543,-67.055,415.507,167.764,41.744,157.754
C07247=1031.538,-67.305,415.518,167.762,41.744,157.754
C07248=1031.531,-67.555,415.530,167.759,41.746,157.754
C07249=1031.525,-67.804,415.541,167.756,41.747,157.754
C07250=1031.519,-68.087,415.554,167.753,41.748,157.754
C07251=1031.512,-68.370,415.567,167.749,41.750,157.754
C07252=1031.505,-68.652,415.581,167.747,41.751,157.754
C07253=1031.498,-68.934,415.594,167.744,41.752,157.754
C07254=1031.492,-69.185,415.605,167.741,41.753,157.754
C07255=1031.486,-69.434,415.616,167.738,41.755,157.755
C07256=1031.479,-69.684,415.628,167.735,41.756,157.755
C07257=1031.474,-69.933,415.639,167.732,41.757,157.755
C07258=1031.467,-70.183,415.650,167.730,41.759,157.755
C07259=1031.462,-70.432,415.662,167.727,41.760,157.755
C07260=1031.456,-70.682,415.673,167.724,41.761,157.755
C07261=1031.450,-70.932,415.684,167.721,41.762,157.755
C07262=1031.444,-71.181,415.696,167.719,41.764,157.755
C07263=1031.438,-71.431,415.707,167.717,41.765,157.755
C07264=1031.433,-71.681,415.719,167.714,41.766,157.755
C07265=1031.426,-71.931,415.730,167.711,41.767,157.755
C07266=1031.420,-72.180,415.741,167.708,41.769,157.755
C07267=1031.414,-72.430,415.753,167.705,41.770,157.755
C07268=1031.408,-72.680,415.763,167.702,41.771,157.755
C07269=1031.402,-72.929,415.775,167.700,41.773,157.755
C07270=1031.396,-73.179,415.787,167.697,41.774,157.755
C07271=1031.391,-73.429,415.798,167.694,41.775,157.755
C07272=1031.384,-73.679,415.809,167.691,41.776,157.755
C07273=1031.378,-73.928,415.821,167.689,41.778,157.755
C07274=1031.373,-74.177,415.831,167.686,41.779,157.755
C07275=1031.366,-74.427,415.843,167.684,41.780,157.756
C07276=1031.361,-74.677,415.854,167.681,41.781,157.756
C07277=1031.354,-74.927,415.865,167.678,41.783,157.756
C07278=1031.348,-75.177,415.876,167.675,41.784,157.756
C07279=1031.343,-75.426,415.887,167.672,41.785,157.756
C07280=1031.336,-75.676,415.897,167.670,41.787,157.756
C07281=1031.330,-75.925,415.908,167.667,41.788,157.756
C07282=1031.324,-76.176,415.919,167.664,41.790,157.756
C07283=1031.318,-76.424,415.931,167.661,41.791,157.756
